// TIA Portal project "FactoryIO_Template_S7-1200_V15_V15.1" (V15.1)
// Vorlageprojekt für das Buch mit Zielsystem S7-1200

(* hardware
DEVICE "S7-1200 station_2"  S7-1200 Station
   slot 0: "Rack_0"  S7-1200 Rack  Rack  V1.0
   slot 1: "PLC_1"  CPU 1215C DC/DC/DC  6ES7 215-1AG40-0XB0  V4.2
   slot 2: "DI 16x24VDC_1"  6ES7 221-1BH32-0XB0  V2.0
   slot 3: "DQ 16x24VDC_1"  SM 1222 DQ16 x 24VDC  6ES7 222-1BH32-0XB0  V2.0
DEVICE "HMI_1"  TP1200 Comfort
   slot 0: "HMI_1"  TP1200 Comfort  6AV2 124-0MC01-0AX0  15.1.0.0
   slot 1: "HMI_RT_1"  TP1200 Comfort  6AV2 124-0MC01-0AX0  15.1.0.0
   slot 5: "HMI_1.IE_CP_1"  PROFINET Interface  15.0.1.0
      slot 1: "PROFINET Interface_1"  PROFINET Interface
         slot 1: "Port_1"  Port
         slot 2: "Port_2"  Port
   slot 7: "HMI_1.MPI/DP_CP_1"  MPI/DP Interface  15.0.1.0
*)

// ===== PLC "PLC_1"  CPU 1215C DC/DC/DC =====

VAR_GLOBAL   // PLC tag table "Default tag table"
   "Green Base Conv_Timer" AT %M5.6 : Bool;
   "Green Lid Conv_Timer" AT %M5.7 : Bool;
   "Metal Base Conv_Timer" AT %M6.0 : Bool;
   "Metal Lid Conv_Timer" AT %M6.1 : Bool;
   "Blue Base Conv_Timer" AT %M6.2 : Bool;
   "Blue Lid Conv_Timer" AT %M6.3 : Bool;
   "RESET_Conv_Timers" AT %M6.4 : Bool;
   "Emitter_Emit" AT %Q4.7 : Bool;
   "Emitter_Part" AT %QD30 : DInt;
   "Counter_Reset" AT %M6.5 : Bool;
   "n_trig[4]" AT %M5.5 : Bool;
   "at load" AT %I13.5 : Bool;
   "left" AT %Q5.2 : Bool;
   "right" AT %Q5.3 : Bool;
   "lift" AT %Q5.4 : Bool;
   "targeted position" AT %QD34 : DInt;
   "at unload" AT %I13.7 : Bool;
   "moving x" AT %I14.0 : Bool;
   "moving z" AT %I14.1 : Bool;
   "at right" AT %I14.2 : Bool;
   "at left" AT %I14.3 : Bool;
   "at middle" AT %I14.4 : Bool;
   "shelf value" AT %MW46 : Word;
   "at entry" AT %I14.5 : Bool;
   "at exit" AT %I14.6 : Bool;
   "entry conveyor(1)" AT %Q5.5 : Bool;
   "loading coneyor" AT %Q5.6 : Bool;
   "unloading coneyor" AT %Q5.7 : Bool;
   "exit conveyor" AT %Q6.0 : Bool;
   "FactoryIo_BugFix" AT %I14.7 : Bool;
   "Box Timing Temp" AT %M6.7 : Bool;
   "Boxes Emitter" AT %Q5.1 : Bool;
   "Boxes Conevyor" AT %Q5.0 : Bool;
   "Product Near Box" AT %I13.6 : Bool;
   "M11" AT %MD60 : DInt;
   "M22" AT %MD64 : DInt;
   "M33" AT %MD68 : DInt;
   "M44" AT %MD72 : DInt;
   "M55" AT %MD76 : DInt;
   "M66" AT %MD80 : DInt;
   "cont sinsor1" AT %I15.0 : Bool;
   "cont sinsor2" AT %I15.1 : Bool;
   "cont sinsor3" AT %I15.2 : Bool;
   "M77" AT %MD88 : DInt;
   "M88" AT %MD92 : DInt;
   "M99" AT %MD96 : DInt;
   "resat" AT %M100.0 : Bool;
   "M110" AT %MD110 : DInt;
   "M120" AT %MD114 : DInt;
   "M130" AT %MD118 : DInt;
   "HMI_UNLOAD" AT %I122.0 : Bool;
END_VAR

VAR_GLOBAL   // PLC tag table "Default tag table_1"
   "ntrig3" AT %M0.4 : Bool;
   "Sorter Memory" AT %MW2 : Word;
   "Metal Base Belt" AT %Q1.1 : Bool;
   "Metal Lid Belt" AT %Q1.2 : Bool;
   "Green Base Belt" AT %Q1.3 : Bool;
   "Green Lid Belt" AT %Q1.4 : Bool;
   "Blue Base Belt" AT %Q1.5 : Bool;
   "Blue Lid Belt" AT %Q1.6 : Bool;
   "#p_trig[0]" AT %M1.7 : Bool;
   "#p_trig[1]" AT %M4.0 : Bool;
   "#p_trig[2]" AT %M4.1 : Bool;
   "#p_trig[3]" AT %M4.2 : Bool;
   "Lid at place" AT %M4.3 : Bool;
   "Lid Clamped" AT %M4.4 : Bool;
   "Two_Axis_Sequence_Done" AT %M4.5 : Bool;
   "Clamp_Lid" AT %M4.6 : Bool;
   "Raise_Lid" AT %M4.7 : Bool;
   "MB_Available" AT %I10.2 : Bool;
   "ML_Available" AT %I10.3 : Bool;
   "GB_Available" AT %I10.4 : Bool;
   "GL_Available" AT %I10.5 : Bool;
   "BB_Available" AT %I10.6 : Bool;
   "BL_Available" AT %I10.7 : Bool;
   "Metal Base Clamp_Positioned" AT %I11.0 : Bool;
   "Metal Lid Clamp_Positioned" AT %I11.1 : Bool;
   "Green Base Clamp_Positioned" AT %I11.2 : Bool;
   "Green Lid Clamp_Positioned" AT %I11.3 : Bool;
   "Blue Base Clamp_Positioned" AT %I11.4 : Bool;
   "Blue Lid Clamp_Positioned" AT %I11.5 : Bool;
   "Metal Lid C_Conv" AT %Q2.5 : Bool;
   "Metal Base C_Conv" AT %Q2.6 : Bool;
   "Green Lid C_Conv" AT %Q2.7 : Bool;
   "Green Base C_Conv" AT %Q3.0 : Bool;
   "Blue Lid C_Conv" AT %Q3.1 : Bool;
   "Blue Base C_Conv" AT %Q3.2 : Bool;
   "Metal Lid (Clamped)" AT %I11.6 : Bool;
   "Metal Base (Clamped)" AT %I11.7 : Bool;
   "Green Lid (Clamped)" AT %I12.0 : Bool;
   "Green Base (Clamped)" AT %I12.1 : Bool;
   "Blue Lid (Clamped)" AT %I12.2 : Bool;
   "Blue Base (Clamped)" AT %I12.3 : Bool;
   "ML (Clamp)" AT %Q1.7 : Bool;
   "MB (Clamp)" AT %Q2.0 : Bool;
   "GL (Clamp)" AT %Q2.1 : Bool;
   "GB (Clamp)" AT %Q2.2 : Bool;
   "BL (Clamp)" AT %Q2.3 : Bool;
   "BB (Clamp)" AT %Q2.4 : Bool;
   "Metal Piece (Raise)" AT %Q3.3 : Bool;
   "Green Piece (Raise)" AT %Q3.4 : Bool;
   "Blue Piece (Raise)" AT %Q3.5 : Bool;
   "Moving X1" AT %I12.4 : Bool;
   "Moving Z1" AT %I12.5 : Bool;
   "Moving X2" AT %I12.6 : Bool;
   "Moving Z2" AT %I12.7 : Bool;
   "Moving X3" AT %I13.0 : Bool;
   "Moving Z3" AT %I13.1 : Bool;
   "Grab1" AT %Q4.4 : Bool;
   "Grab2" AT %Q4.5 : Bool;
   "Grab3" AT %Q4.6 : Bool;
   "Move X1" AT %Q3.6 : Bool;
   "Move Z1" AT %Q3.7 : Bool;
   "Move X2" AT %Q4.0 : Bool;
   "Move Z2" AT %Q4.1 : Bool;
   "Move X3" AT %Q4.2 : Bool;
   "Move Z3" AT %Q4.3 : Bool;
   "Two_Axis_Sequence_Done1" AT %M0.5 : Bool;
   "Two_Axis_Sequence_Done2" AT %M0.6 : Bool;
   "Two_Axis_Sequence_Done3" AT %M0.7 : Bool;
   "Item_Detected1" AT %I13.2 : Bool;
   "Item_Detected2" AT %I13.3 : Bool;
   "Item_Detected3" AT %I13.4 : Bool;
   "ML C Latch" AT %M1.0 : Bool;
   "MB C Latch" AT %M1.1 : Bool;
   "GL C Latch" AT %M1.2 : Bool;
   "GB C Latch" AT %M1.3 : Bool;
   "BL C Latch" AT %M1.4 : Bool;
   "BB C Latch" AT %M1.5 : Bool;
   "RESET_METAL" AT %M1.6 : Bool;
   "RESET_GREEN" AT %M5.0 : Bool;
   "RESET_BLUE" AT %M5.1 : Bool;
   "Tag_1" AT %M10.7 : Bool;
   "Tag_2" AT %M5.3 : Bool;
   "Tag_3" AT %M5.4 : Bool;
END_VAR

VAR_GLOBAL CONSTANT   // PLC tag table "Default tag table_1"
   "None(1)" : Pip := 65535;
   "Automatic update(1)" : Pip := 0;
   "PIP 1(1)" : Pip := 1;
   "PIP 2(1)" : Pip := 2;
   "PIP 3(1)" : Pip := 3;
   "PIP 4(1)" : Pip := 4;
   "PIP OB Servo(1)" : Pip := 32768;
   "Local~MC(2)" : Hw_SubModule := 51;
   "Local~Common(2)" : Hw_SubModule := 50;
   "Local~Device(2)" : Hw_Device := 32;
   "Local~Configuration(2)" : Hw_SubModule := 33;
   "Local~Exec(2)" : Hw_SubModule := 52;
   "Local(2)" : Hw_SubModule := 49;
   "Local~PROFINET_interface_1(1)" : Hw_Interface := 64;
   "Local~PROFINET_interface_1~Port_1(1)" : Hw_Interface := 65;
   "Local~PROFINET_interface_1~Port_2(1)" : Hw_Interface := 66;
   "Local~HSC_1(2)" : Hw_Hsc := 257;
   "Local~HSC_2(2)" : Hw_Hsc := 258;
   "Local~HSC_3(2)" : Hw_Hsc := 259;
   "Local~HSC_4(2)" : Hw_Hsc := 260;
   "Local~HSC_5(2)" : Hw_Hsc := 261;
   "Local~HSC_6(2)" : Hw_Hsc := 262;
   "Local~AI_2_AQ_2_1(1)" : Hw_SubModule := 263;
   "Local~DI_14_DQ_10_1(1)" : Hw_SubModule := 264;
   "Local~Pulse_1(2)" : Hw_Pwm := 265;
   "Local~Pulse_2(2)" : Hw_Pwm := 266;
   "Local~Pulse_3(2)" : Hw_Pwm := 267;
   "Local~Pulse_4(2)" : Hw_Pwm := 268;
   "OB_Main(2)" : OB_PCYCLE := 1;
   "Local~DI_16x24VDC_1(1)" : Hw_SubModule := 269;
   "Local~DQ_8x24VDC__1" : Hw_SubModule := 270;
END_VAR

VAR_GLOBAL   // PLC tag table "Standard-Variablentabelle"
   "Entry Conveyor Stop" AT %M0.0 : Bool;
   "ntrig0" AT %M0.1 : Bool;
   "Stop Sensor 1" AT %I10.0 : Bool;
   "Stop Sensor 2" AT %I10.1 : Bool;
   "ntrig1" AT %M0.2 : Bool;
   "Sorting Conveyor 1" AT %Q0.7 : Bool;
   "Sorting Conveyor 2" AT %Q1.0 : Bool;
   "ntrig2" AT %M0.3 : Bool;
END_VAR

VAR_GLOBAL CONSTANT   // PLC tag table "Standard-Variablentabelle"
   "Keiner" : Pip := 65535;
   "Automatische Aktualisierung" : Pip := 0;
   "TPA 1" : Pip := 1;
   "TPA 2" : Pip := 2;
   "TPA 3" : Pip := 3;
   "TPA 4" : Pip := 4;
   "TPA OB Servo" : Pip := 32768;
   "Local~MC(1)" : Hw_SubModule := 51;
   "Local~Common(1)" : Hw_SubModule := 50;
   "Local~Device(1)" : Hw_Device := 32;
   "Local~Configuration(1)" : Hw_SubModule := 33;
   "Local~Exec(1)" : Hw_SubModule := 52;
   "Local(1)" : Hw_SubModule := 49;
   "Local~PROFINET-Schnittstelle_1" : Hw_Interface := 64;
   "Local~PROFINET-Schnittstelle_1~Port_1" : Hw_Interface := 65;
   "Local~HSC_1(1)" : Hw_Hsc := 257;
   "Local~HSC_2(1)" : Hw_Hsc := 258;
   "Local~HSC_3(1)" : Hw_Hsc := 259;
   "Local~HSC_4(1)" : Hw_Hsc := 260;
   "Local~HSC_5(1)" : Hw_Hsc := 261;
   "Local~HSC_6(1)" : Hw_Hsc := 262;
   "Local~AI_2_1" : Hw_SubModule := 263;
   "Local~DI_6_DQ_4_1" : Hw_SubModule := 264;
   "Local~Pulse_1(1)" : Hw_Pwm := 265;
   "Local~Pulse_2(1)" : Hw_Pwm := 266;
   "Local~Pulse_3(1)" : Hw_Pwm := 267;
   "Local~Pulse_4(1)" : Hw_Pwm := 268;
   "OB_Main(1)" : OB_PCYCLE := 1;
END_VAR

VAR_GLOBAL   // PLC tag table "Tag table from XML_1"
   "Entry Conveyor" AT %Q0.0 : Bool;
   "Metal Base Arm" AT %Q0.1 : Bool;
   "Metal Lid Arm" AT %Q0.2 : Bool;
   "Green Base Arm" AT %Q0.3 : Bool;
   "Green Lid Arm" AT %Q0.4 : Bool;
   "Blue Base Arm" AT %Q0.5 : Bool;
   "Blue Lid Arm" AT %Q0.6 : Bool;
   "Vision Sensor 1 (Value)" AT %ID30 : DInt;
END_VAR

DATA_BLOCK "Pick&Place_DB"   // DB2
{ S7_Optimized_Access := 'TRUE' }
VERSION : 0.1
// stored: InstanceOfName Pick&Place
"Pick&Place"
BEGIN
END_DATA_BLOCK

DATA_BLOCK "Base_Conveyor_DB"   // DB3
{ S7_Optimized_Access := 'TRUE' }
VERSION : 0.1
// stored: InstanceOfName Base_Conveyor
"Base_Conveyor"
BEGIN
END_DATA_BLOCK

DATA_BLOCK "Base_Conveyor_DB_1"   // DB4
{ S7_Optimized_Access := 'TRUE' }
VERSION : 0.1
// stored: InstanceOfName Base_Conveyor
"Base_Conveyor"
BEGIN
END_DATA_BLOCK

DATA_BLOCK "Base_Conveyor_DB_2"   // DB5
{ S7_Optimized_Access := 'TRUE' }
VERSION : 0.1
// stored: InstanceOfName Base_Conveyor
"Base_Conveyor"
BEGIN
END_DATA_BLOCK

DATA_BLOCK "Lids_Conveyor_DB"   // DB6
{ S7_Optimized_Access := 'TRUE' }
VERSION : 0.1
// stored: InstanceOfName Lids_Conveyor
"Lids_Conveyor"
BEGIN
END_DATA_BLOCK

DATA_BLOCK "Lids_Conveyor_DB_1"   // DB7
{ S7_Optimized_Access := 'TRUE' }
VERSION : 0.1
// stored: InstanceOfName Lids_Conveyor
"Lids_Conveyor"
BEGIN
END_DATA_BLOCK

DATA_BLOCK "Lids_Conveyor_DB_2"   // DB8
{ S7_Optimized_Access := 'TRUE' }
VERSION : 0.1
// stored: InstanceOfName Lids_Conveyor
"Lids_Conveyor"
BEGIN
END_DATA_BLOCK

DATA_BLOCK "Clamp_Base1"   // DB9
{ S7_Optimized_Access := 'TRUE' }
VERSION : 0.1
// stored: InstanceOfName Clamp
"Clamp"
BEGIN
END_DATA_BLOCK

DATA_BLOCK "Clamp_Base2"   // DB10
{ S7_Optimized_Access := 'TRUE' }
VERSION : 0.1
// stored: InstanceOfName Clamp
"Clamp"
BEGIN
END_DATA_BLOCK

DATA_BLOCK "Clamp_Base3"   // DB11
{ S7_Optimized_Access := 'TRUE' }
VERSION : 0.1
// stored: InstanceOfName Clamp
"Clamp"
BEGIN
END_DATA_BLOCK

DATA_BLOCK "Clamp_lid1"   // DB12
{ S7_Optimized_Access := 'TRUE' }
VERSION : 0.1
// stored: InstanceOfName Clamp
"Clamp"
BEGIN
END_DATA_BLOCK

DATA_BLOCK "Clamp_lid2"   // DB13
{ S7_Optimized_Access := 'TRUE' }
VERSION : 0.1
// stored: InstanceOfName Clamp
"Clamp"
BEGIN
END_DATA_BLOCK

DATA_BLOCK "Clamp_lid3"   // DB14
{ S7_Optimized_Access := 'TRUE' }
VERSION : 0.1
// stored: InstanceOfName Clamp
"Clamp"
BEGIN
END_DATA_BLOCK

DATA_BLOCK "Pick&Place_DB_1"   // DB15
{ S7_Optimized_Access := 'TRUE' }
VERSION : 0.1
// stored: InstanceOfName Pick&Place
"Pick&Place"
BEGIN
END_DATA_BLOCK

DATA_BLOCK "Pick&Place_DB_2"   // DB16
{ S7_Optimized_Access := 'TRUE' }
VERSION : 0.1
// stored: InstanceOfName Pick&Place
"Pick&Place"
BEGIN
END_DATA_BLOCK

DATA_BLOCK "Pick&Place_DB_3"   // DB17
{ S7_Optimized_Access := 'TRUE' }
VERSION : 0.1
// stored: InstanceOfName Pick&Place
"Pick&Place"
BEGIN
END_DATA_BLOCK

DATA_BLOCK "Block_1_DB"   // DB24
{ S7_Optimized_Access := 'TRUE' }
VERSION : 0.1
// stored: InstanceOfName Block_1
"Block_1"
BEGIN
END_DATA_BLOCK

DATA_BLOCK "Block_1_DB_1"   // DB25
{ S7_Optimized_Access := 'TRUE' }
VERSION : 0.1
// stored: InstanceOfName Block_1
"Block_1"
BEGIN
END_DATA_BLOCK

DATA_BLOCK "Block_2_DB"   // DB26
{ S7_Optimized_Access := 'TRUE' }
VERSION : 0.1
// stored: InstanceOfName Block_2
"Block_2"
BEGIN
END_DATA_BLOCK

DATA_BLOCK "Block_1_DB_2"   // DB27
{ S7_Optimized_Access := 'TRUE' }
VERSION : 0.1
// stored: InstanceOfName Block_1
"Block_1"
BEGIN
END_DATA_BLOCK

// folder: System blocks/Program resources

DATA_BLOCK "IEC_Timer_0_DB"   // DB1
{ S7_Optimized_Access := 'TRUE' }
AUTHOR : Simatic
FAMILY : IEC
NAME : IEC_TMR
VERSION : 1.0
// stored: InstanceOfName IEC_TIMER
"IEC_TIMER"
BEGIN
END_DATA_BLOCK

DATA_BLOCK "IEC_Timer_0_DB_1"   // DB18
{ S7_Optimized_Access := 'TRUE' }
AUTHOR : Simatic
FAMILY : IEC
NAME : IEC_TMR
VERSION : 1.0
// stored: InstanceOfName IEC_TIMER
"IEC_TIMER"
BEGIN
END_DATA_BLOCK

DATA_BLOCK "IEC_Timer_0_DB_2"   // DB19
{ S7_Optimized_Access := 'TRUE' }
AUTHOR : Simatic
FAMILY : IEC
NAME : IEC_TMR
VERSION : 1.0
// stored: InstanceOfName IEC_TIMER
"IEC_TIMER"
BEGIN
END_DATA_BLOCK

DATA_BLOCK "IEC_Timer_0_DB_3"   // DB20
{ S7_Optimized_Access := 'TRUE' }
AUTHOR : Simatic
FAMILY : IEC
NAME : IEC_TMR
VERSION : 1.0
// stored: InstanceOfName IEC_TIMER
"IEC_TIMER"
BEGIN
END_DATA_BLOCK

DATA_BLOCK "IEC_Timer_0_DB_4"   // DB21
{ S7_Optimized_Access := 'TRUE' }
AUTHOR : Simatic
FAMILY : IEC
NAME : IEC_TMR
VERSION : 1.0
// stored: InstanceOfName IEC_TIMER
"IEC_TIMER"
BEGIN
END_DATA_BLOCK

DATA_BLOCK "IEC_Timer_0_DB_5"   // DB22
{ S7_Optimized_Access := 'TRUE' }
AUTHOR : Simatic
FAMILY : IEC
NAME : IEC_TMR
VERSION : 1.0
// stored: InstanceOfName IEC_TIMER
"IEC_TIMER"
BEGIN
END_DATA_BLOCK

DATA_BLOCK "IEC_Counter_0_DB[1]"   // DB23
{ S7_Optimized_Access := 'TRUE' }
AUTHOR : Simatic
FAMILY : IEC
NAME : CNTR
VERSION : 1.0
// stored: InstanceOfName IEC_COUNTER
"IEC_COUNTER"
BEGIN
END_DATA_BLOCK

DATA_BLOCK "IEC_Timer_0_DB_6"   // DB28
{ S7_Optimized_Access := 'TRUE' }
AUTHOR : Simatic
FAMILY : IEC
NAME : IEC_TMR
VERSION : 1.0
// stored: InstanceOfName IEC_TIMER
"IEC_TIMER"
BEGIN
END_DATA_BLOCK

DATA_BLOCK "IEC_Counter_0_DB"   // DB29
{ S7_Optimized_Access := 'TRUE' }
AUTHOR : Simatic
FAMILY : IEC
NAME : CNTR
VERSION : 1.0
// stored: InstanceOfName IEC_COUNTER
"IEC_COUNTER"
BEGIN
END_DATA_BLOCK

DATA_BLOCK "IEC_Counter_0_DB_1"   // DB30
{ S7_Optimized_Access := 'TRUE' }
AUTHOR : Simatic
FAMILY : IEC
NAME : CNTR
VERSION : 1.0
// stored: InstanceOfName IEC_COUNTER
"IEC_COUNTER"
BEGIN
END_DATA_BLOCK

DATA_BLOCK "IEC_Counter_0_DB_2"   // DB31
{ S7_Optimized_Access := 'TRUE' }
AUTHOR : Simatic
FAMILY : IEC
NAME : CNTR
VERSION : 1.0
// stored: InstanceOfName IEC_COUNTER
"IEC_COUNTER"
BEGIN
END_DATA_BLOCK

DATA_BLOCK "IEC_Counter_0_DB_3"   // DB32
{ S7_Optimized_Access := 'TRUE' }
AUTHOR : Simatic
FAMILY : IEC
NAME : CNTR
VERSION : 1.0
// stored: InstanceOfName IEC_COUNTER
"IEC_COUNTER"
BEGIN
END_DATA_BLOCK

DATA_BLOCK "IEC_Counter_0_DB_4"   // DB33
{ S7_Optimized_Access := 'TRUE' }
AUTHOR : Simatic
FAMILY : IEC
NAME : CNTR
VERSION : 1.0
// stored: InstanceOfName IEC_COUNTER
"IEC_COUNTER"
BEGIN
END_DATA_BLOCK

DATA_BLOCK "IEC_Counter_0_DB_5"   // DB34
{ S7_Optimized_Access := 'TRUE' }
AUTHOR : Simatic
FAMILY : IEC
NAME : CNTR
VERSION : 1.0
// stored: InstanceOfName IEC_COUNTER
"IEC_COUNTER"
BEGIN
END_DATA_BLOCK

DATA_BLOCK "IEC_Counter_0_DB_6"   // DB35
{ S7_Optimized_Access := 'TRUE' }
AUTHOR : Simatic
FAMILY : IEC
NAME : CNTR
VERSION : 1.0
// stored: InstanceOfName IEC_COUNTER
"IEC_COUNTER"
BEGIN
END_DATA_BLOCK

DATA_BLOCK "IEC_Counter_0_DB_7"   // DB36
{ S7_Optimized_Access := 'TRUE' }
AUTHOR : Simatic
FAMILY : IEC
NAME : CNTR
VERSION : 1.0
// stored: InstanceOfName IEC_COUNTER
"IEC_COUNTER"
BEGIN
END_DATA_BLOCK

DATA_BLOCK "IEC_Counter_0_DB_8"   // DB37
{ S7_Optimized_Access := 'TRUE' }
AUTHOR : Simatic
FAMILY : IEC
NAME : CNTR
VERSION : 1.0
// stored: InstanceOfName IEC_COUNTER
"IEC_COUNTER"
BEGIN
END_DATA_BLOCK

DATA_BLOCK "IEC_Counter_0_DB_9"   // DB38
{ S7_Optimized_Access := 'TRUE' }
AUTHOR : Simatic
FAMILY : IEC
NAME : CNTR
VERSION : 1.0
// stored: InstanceOfName IEC_COUNTER
"IEC_COUNTER"
BEGIN
END_DATA_BLOCK

DATA_BLOCK "IEC_Counter_0_DB_10"   // DB39
{ S7_Optimized_Access := 'TRUE' }
AUTHOR : Simatic
FAMILY : IEC
NAME : CNTR
VERSION : 1.0
// stored: InstanceOfName IEC_COUNTER
"IEC_COUNTER"
BEGIN
END_DATA_BLOCK

// folder: (top level)

FUNCTION_BLOCK "Clamp"   // FB1, LAD
{ S7_Optimized_Access := 'TRUE' }
VERSION : 0.1
   VAR_INPUT
      Start_Clamper_Sequence : Bool;
      Clamped_Sensor : Bool;
      Axis_Seq_Done : Bool;
   END_VAR
   VAR_OUTPUT
      Clamp : Bool;
      Raise_Clamp : Bool;
      Sequence_Done : Bool;
   END_VAR
   VAR
      Sequence_Active : Bool;
      Step1 : Int;
   END_VAR
   VAR RETAIN
      "TimeOn1.PT" : Int;
   END_VAR
   VAR
      "p_trig[1]" : Bool;
      "p_trig[0]" : Bool;
      "p_trig[2]" : Bool;
      "p_trig[3]" : Bool;
      Sequence_Done_Pulse : Bool;
      IEC_Timer_0_Instance : TON_TIME;
   END_VAR
   VAR_TEMP   // added for the SCL form of the ladder/FBD networks
      _w1 : Bool;
      _w2 : Bool;
      _w3 : Bool;
   END_VAR
BEGIN

REGION Network 1
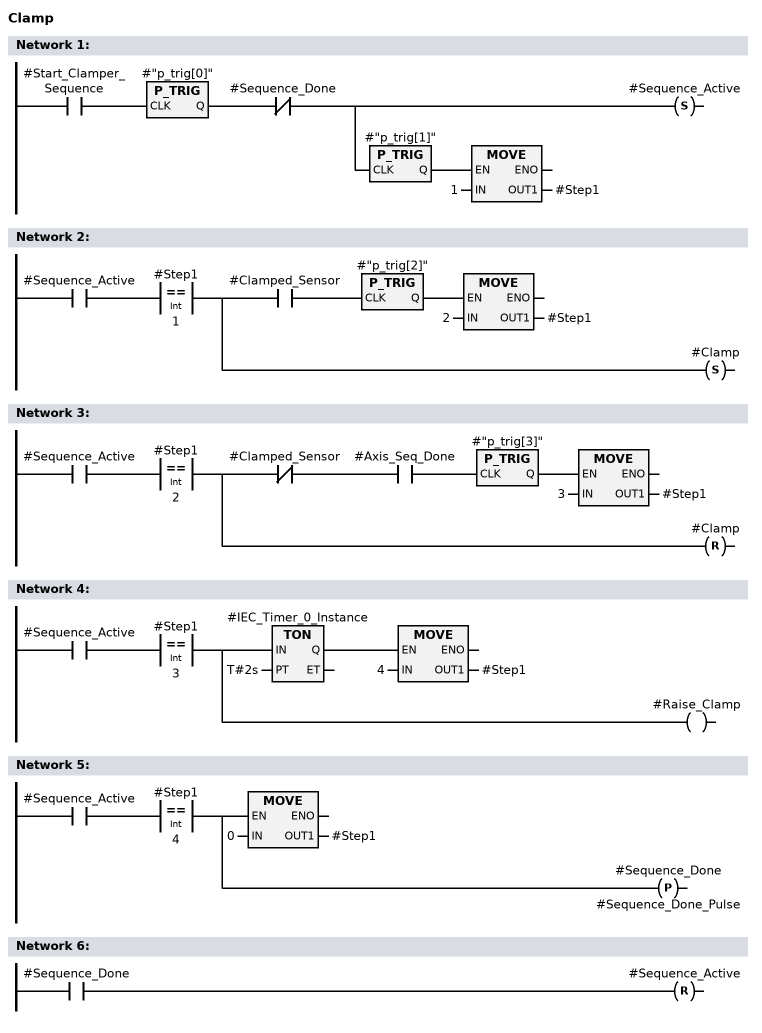
   RUNG wire#powerrail
      Contact( #Start_Clamper_Sequence )
      P_Trig( #"p_trig[0]" )
      I_Contact( #Sequence_Done )
      wire#w1
      S_Coil( #Sequence_Active )
   END_RUNG
   RUNG wire#w1
      P_Trig( #"p_trig[1]" )
      Move(in := 1, out1 => #Step1)
   END_RUNG
   // the same network as SCL:
   #_w1 := #Start_Clamper_Sequence AND NOT #"p_trig[0]";   // rising edge
   #"p_trig[0]" := #Start_Clamper_Sequence;
   #_w2 := #_w1 AND NOT #Sequence_Done;
   IF #_w2 THEN #Sequence_Active := TRUE; END_IF;
   #_w3 := #_w2 AND NOT #"p_trig[1]";   // rising edge
   #"p_trig[1]" := #_w2;
   IF #_w3 THEN #Step1 := 1; END_IF;
END_REGION

REGION Network 2
   RUNG wire#powerrail
      Contact( #Sequence_Active )
      { S7_Templates := "SrcType := Int" } EQ_Contact(in1 := #Step1, in2 := 1)
      wire#w1
      Contact( #Clamped_Sensor )
      P_Trig( #"p_trig[2]" )
      Move(in := 2, out1 => #Step1)
   END_RUNG
   RUNG wire#w1
      S_Coil( #Clamp )
   END_RUNG
   // the same network as SCL:
   #_w1 := #Sequence_Active AND (#Step1 = 1);
   #_w2 := #_w1 AND #Clamped_Sensor;
   #_w3 := #_w2 AND NOT #"p_trig[2]";   // rising edge
   #"p_trig[2]" := #_w2;
   IF #_w3 THEN #Step1 := 2; END_IF;
   IF #_w1 THEN #Clamp := TRUE; END_IF;
END_REGION

REGION Network 3
   RUNG wire#powerrail
      Contact( #Sequence_Active )
      { S7_Templates := "SrcType := Int" } EQ_Contact(in1 := #Step1, in2 := 2)
      wire#w1
      I_Contact( #Clamped_Sensor )
      Contact( #Axis_Seq_Done )
      P_Trig( #"p_trig[3]" )
      Move(in := 3, out1 => #Step1)
   END_RUNG
   RUNG wire#w1
      R_Coil( #Clamp )
   END_RUNG
   // the same network as SCL:
   #_w1 := #Sequence_Active AND (#Step1 = 2);
   #_w2 := #_w1 AND NOT #Clamped_Sensor AND #Axis_Seq_Done;
   #_w3 := #_w2 AND NOT #"p_trig[3]";   // rising edge
   #"p_trig[3]" := #_w2;
   IF #_w3 THEN #Step1 := 3; END_IF;
   IF #_w1 THEN #Clamp := FALSE; END_IF;
END_REGION

REGION Network 4
   #_w1 := #Sequence_Active AND (#Step1 = 3);
   #IEC_Timer_0_Instance(IN := #_w1, PT := T#2s);   // TON
   IF #IEC_Timer_0_Instance.Q THEN #Step1 := 4; END_IF;
   #Raise_Clamp := #_w1;
END_REGION

REGION Network 5
   #_w1 := #Sequence_Active AND (#Step1 = 4);
   IF #_w1 THEN #Step1 := 0; END_IF;
   #Sequence_Done := #_w1 AND NOT #Sequence_Done_Pulse;   // rising edge
   #Sequence_Done_Pulse := #_w1;
END_REGION

REGION Network 6
   RUNG wire#powerrail
      Contact( #Sequence_Done )
      R_Coil( #Sequence_Active )
   END_RUNG
   // the same network as SCL:
   IF #Sequence_Done THEN #Sequence_Active := FALSE; END_IF;
END_REGION
END_FUNCTION_BLOCK

FUNCTION_BLOCK "Pick&Place"   // FB2, LAD
{ S7_Optimized_Access := 'TRUE' }
VERSION : 0.1
   VAR_INPUT
      Start_Axis_Sequence : Bool;
      Moving_X : Bool;
      Moving_Z : Bool;
      Item_Detected : Bool;
   END_VAR
   VAR_OUTPUT
      Move_X : Bool;
      Move_Z : Bool;
      Item_Grab : Bool;
      RESET_CLAMP_COND : Bool;
      Sequence_Done : Bool;
   END_VAR
   VAR
      "n_trig[2]" : Bool;
      "n_trig[0]" : Bool;
      "n_trig[1]" : Bool;
      "Step" : Int;
      Sequence_Active : Bool;
      "p_trig[0]" : Bool;
      "p_trig[1]" : Bool;
      "p_trig[2]" : Bool;
      "n_trig[3]" : Bool;
      Sequence_Done_Pulses : Bool;
      "n_trig[4]" : Bool;
   END_VAR
   VAR_TEMP   // added for the SCL form of the ladder/FBD networks
      _w1 : Bool;
      _w2 : Bool;
      _w3 : Bool;
   END_VAR
BEGIN

REGION Network 1
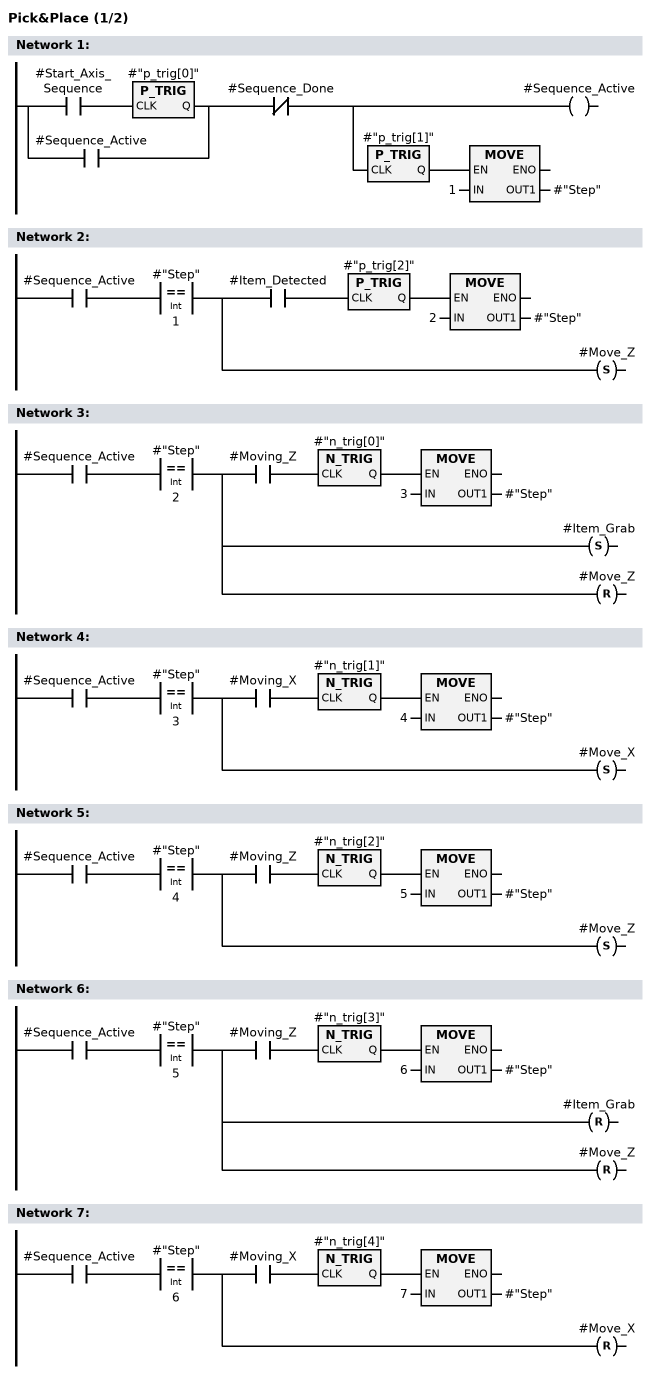
   RUNG wire#powerrail
      Contact( #Start_Axis_Sequence )
      P_Trig( #"p_trig[0]" )
      wire#w1
      I_Contact( #Sequence_Done )
      wire#w2
      Coil( #Sequence_Active )
   END_RUNG
   RUNG wire#powerrail
      Contact( #Sequence_Active )
   END_RUNG wire#w1
   RUNG wire#w2
      P_Trig( #"p_trig[1]" )
      Move(in := 1, out1 => #"Step")
   END_RUNG
   // the same network as SCL:
   #_w1 := #Start_Axis_Sequence AND NOT #"p_trig[0]";   // rising edge
   #"p_trig[0]" := #Start_Axis_Sequence;
   #Sequence_Active := (#_w1 OR #Sequence_Active) AND NOT #Sequence_Done;
   #_w2 := #Sequence_Active AND NOT #"p_trig[1]";   // rising edge
   #"p_trig[1]" := #Sequence_Active;
   IF #_w2 THEN #"Step" := 1; END_IF;
END_REGION

REGION Network 2
   RUNG wire#powerrail
      Contact( #Sequence_Active )
      { S7_Templates := "SrcType := Int" } EQ_Contact(in1 := #"Step", in2 := 1)
      wire#w1
      Contact( #Item_Detected )
      P_Trig( #"p_trig[2]" )
      Move(in := 2, out1 => #"Step")
   END_RUNG
   RUNG wire#w1
      S_Coil( #Move_Z )
   END_RUNG
   // the same network as SCL:
   #_w1 := #Sequence_Active AND (#"Step" = 1);
   #_w2 := #_w1 AND #Item_Detected;
   #_w3 := #_w2 AND NOT #"p_trig[2]";   // rising edge
   #"p_trig[2]" := #_w2;
   IF #_w3 THEN #"Step" := 2; END_IF;
   IF #_w1 THEN #Move_Z := TRUE; END_IF;
END_REGION

REGION Network 3
   RUNG wire#powerrail
      Contact( #Sequence_Active )
      { S7_Templates := "SrcType := Int" } EQ_Contact(in1 := #"Step", in2 := 2)
      wire#w1
      Contact( #Moving_Z )
      N_Trig( #"n_trig[0]" )
      Move(in := 3, out1 => #"Step")
   END_RUNG
   RUNG wire#w1
      S_Coil( #Item_Grab )
   END_RUNG
   RUNG wire#w1
      R_Coil( #Move_Z )
   END_RUNG
   // the same network as SCL:
   #_w1 := #Sequence_Active AND (#"Step" = 2);
   #_w2 := #_w1 AND #Moving_Z;
   #_w3 := NOT #_w2 AND #"n_trig[0]";   // falling edge
   #"n_trig[0]" := #_w2;
   IF #_w3 THEN #"Step" := 3; END_IF;
   IF #_w1 THEN
       #Item_Grab := TRUE;
       #Move_Z := FALSE;
   END_IF;
END_REGION

REGION Network 4
   RUNG wire#powerrail
      Contact( #Sequence_Active )
      { S7_Templates := "SrcType := Int" } EQ_Contact(in1 := #"Step", in2 := 3)
      wire#w1
      Contact( #Moving_X )
      N_Trig( #"n_trig[1]" )
      Move(in := 4, out1 => #"Step")
   END_RUNG
   RUNG wire#w1
      S_Coil( #Move_X )
   END_RUNG
   // the same network as SCL:
   #_w1 := #Sequence_Active AND (#"Step" = 3);
   #_w2 := #_w1 AND #Moving_X;
   #_w3 := NOT #_w2 AND #"n_trig[1]";   // falling edge
   #"n_trig[1]" := #_w2;
   IF #_w3 THEN #"Step" := 4; END_IF;
   IF #_w1 THEN #Move_X := TRUE; END_IF;
END_REGION

REGION Network 5
   RUNG wire#powerrail
      Contact( #Sequence_Active )
      { S7_Templates := "SrcType := Int" } EQ_Contact(in1 := #"Step", in2 := 4)
      wire#w1
      Contact( #Moving_Z )
      N_Trig( #"n_trig[2]" )
      Move(in := 5, out1 => #"Step")
   END_RUNG
   RUNG wire#w1
      S_Coil( #Move_Z )
   END_RUNG
   // the same network as SCL:
   #_w1 := #Sequence_Active AND (#"Step" = 4);
   #_w2 := #_w1 AND #Moving_Z;
   #_w3 := NOT #_w2 AND #"n_trig[2]";   // falling edge
   #"n_trig[2]" := #_w2;
   IF #_w3 THEN #"Step" := 5; END_IF;
   IF #_w1 THEN #Move_Z := TRUE; END_IF;
END_REGION

REGION Network 6
   RUNG wire#powerrail
      Contact( #Sequence_Active )
      { S7_Templates := "SrcType := Int" } EQ_Contact(in1 := #"Step", in2 := 5)
      wire#w1
      Contact( #Moving_Z )
      N_Trig( #"n_trig[3]" )
      Move(in := 6, out1 => #"Step")
   END_RUNG
   RUNG wire#w1
      R_Coil( #Item_Grab )
   END_RUNG
   RUNG wire#w1
      R_Coil( #Move_Z )
   END_RUNG
   // the same network as SCL:
   #_w1 := #Sequence_Active AND (#"Step" = 5);
   #_w2 := #_w1 AND #Moving_Z;
   #_w3 := NOT #_w2 AND #"n_trig[3]";   // falling edge
   #"n_trig[3]" := #_w2;
   IF #_w3 THEN #"Step" := 6; END_IF;
   IF #_w1 THEN
       #Item_Grab := FALSE;
       #Move_Z := FALSE;
   END_IF;
END_REGION

REGION Network 7
   RUNG wire#powerrail
      Contact( #Sequence_Active )
      { S7_Templates := "SrcType := Int" } EQ_Contact(in1 := #"Step", in2 := 6)
      wire#w1
      Contact( #Moving_X )
      N_Trig( #"n_trig[4]" )
      Move(in := 7, out1 => #"Step")
   END_RUNG
   RUNG wire#w1
      R_Coil( #Move_X )
   END_RUNG
   // the same network as SCL:
   #_w1 := #Sequence_Active AND (#"Step" = 6);
   #_w2 := #_w1 AND #Moving_X;
   #_w3 := NOT #_w2 AND #"n_trig[4]";   // falling edge
   #"n_trig[4]" := #_w2;
   IF #_w3 THEN #"Step" := 7; END_IF;
   IF #_w1 THEN #Move_X := FALSE; END_IF;
END_REGION

REGION Network 8
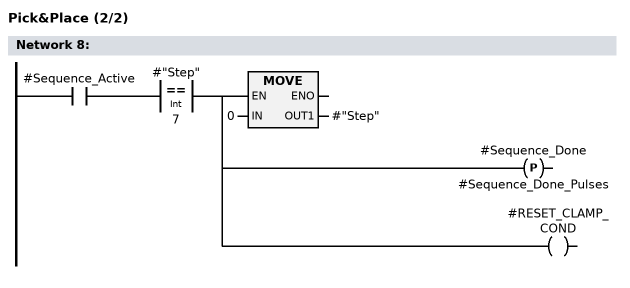
   #_w1 := #Sequence_Active AND (#"Step" = 7);
   IF #_w1 THEN #"Step" := 0; END_IF;
   #Sequence_Done := #_w1 AND NOT #Sequence_Done_Pulses;   // rising edge
   #Sequence_Done_Pulses := #_w1;
   #RESET_CLAMP_COND := #_w1;
END_REGION
END_FUNCTION_BLOCK

FUNCTION_BLOCK "Base_Conveyor"   // FB3, LAD
{ S7_Optimized_Access := 'TRUE' }
VERSION : 0.1
   VAR_INPUT
      Start_Bases_Conveyor : Bool;
      Stop_Bases_Conveyor : Bool;
   END_VAR
   VAR_OUTPUT
      Bases_Conveyor_Active : Bool;
   END_VAR
   VAR_TEMP
      "p_trig[0]" : Bool;
      "n_trig[0]" : Bool;
   END_VAR
   VAR_TEMP   // added for the SCL form of the ladder/FBD networks
      _w1 : Bool;
   END_VAR
BEGIN

REGION Network 1
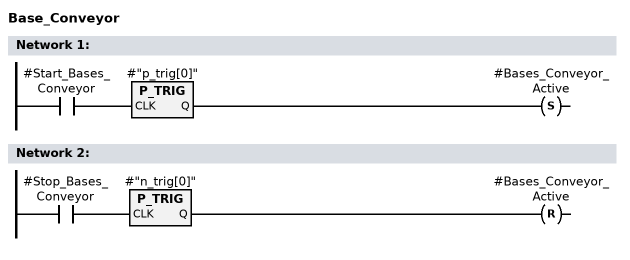
   RUNG wire#powerrail
      Contact( #Start_Bases_Conveyor )
      P_Trig( #"p_trig[0]" )
      S_Coil( #Bases_Conveyor_Active )
   END_RUNG
   // the same network as SCL:
   #_w1 := #Start_Bases_Conveyor AND NOT #"p_trig[0]";   // rising edge
   #"p_trig[0]" := #Start_Bases_Conveyor;
   IF #_w1 THEN #Bases_Conveyor_Active := TRUE; END_IF;
END_REGION

REGION Network 2
   RUNG wire#powerrail
      Contact( #Stop_Bases_Conveyor )
      P_Trig( #"n_trig[0]" )
      R_Coil( #Bases_Conveyor_Active )
   END_RUNG
   // the same network as SCL:
   #_w1 := #Stop_Bases_Conveyor AND NOT #"n_trig[0]";   // rising edge
   #"n_trig[0]" := #Stop_Bases_Conveyor;
   IF #_w1 THEN #Bases_Conveyor_Active := FALSE; END_IF;
END_REGION
END_FUNCTION_BLOCK

FUNCTION_BLOCK "Lids_Conveyor"   // FB4, LAD
{ S7_Optimized_Access := 'TRUE' }
VERSION : 0.1
   VAR_INPUT
      Start_Lids_Conveyor : Bool;
      Stop_Lids_Conveyor : Bool;
   END_VAR
   VAR_OUTPUT
      Lids_Conveyor_Active : Bool;
   END_VAR
   VAR_TEMP
      "p_trig[0]" : Bool;
      "n_trig[0]" : Bool;
   END_VAR
   VAR_TEMP   // added for the SCL form of the ladder/FBD networks
      _w1 : Bool;
   END_VAR
BEGIN

REGION Network 1
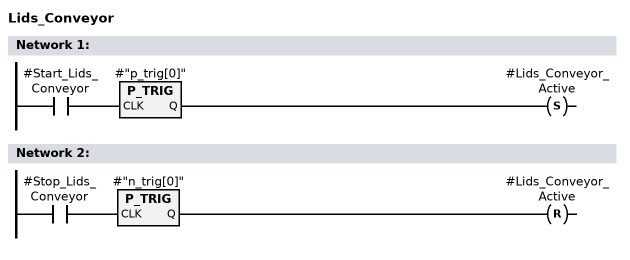
   RUNG wire#powerrail
      Contact( #Start_Lids_Conveyor )
      P_Trig( #"p_trig[0]" )
      S_Coil( #Lids_Conveyor_Active )
   END_RUNG
   // the same network as SCL:
   #_w1 := #Start_Lids_Conveyor AND NOT #"p_trig[0]";   // rising edge
   #"p_trig[0]" := #Start_Lids_Conveyor;
   IF #_w1 THEN #Lids_Conveyor_Active := TRUE; END_IF;
END_REGION

REGION Network 2
   RUNG wire#powerrail
      Contact( #Stop_Lids_Conveyor )
      P_Trig( #"n_trig[0]" )
      R_Coil( #Lids_Conveyor_Active )
   END_RUNG
   // the same network as SCL:
   #_w1 := #Stop_Lids_Conveyor AND NOT #"n_trig[0]";   // rising edge
   #"n_trig[0]" := #Stop_Lids_Conveyor;
   IF #_w1 THEN #Lids_Conveyor_Active := FALSE; END_IF;
END_REGION
END_FUNCTION_BLOCK

FUNCTION_BLOCK "Block_1"   // FB5, LAD
TITLE = stacker crane
{ S7_Optimized_Access := 'TRUE' }
VERSION : 0.1
   VAR_INPUT
      Start_Load_Sequence : Bool;
      Start_Unload_Sequence : Bool;
      "at right" : Bool;
      at_left : Bool;
      "at middle" : Bool;
      "moving X" : Bool;
      "moving Z" : Bool;
   END_VAR
   VAR_OUTPUT
      Stored_Shelf_Value : Int;
      forks_left : Bool;
      forks_right : Bool;
      lift : Bool;
      Unload_Sequence_Done : Bool;
      Load_Sequence_Done : Bool;
      target_position : Int;
   END_VAR
   VAR
      "n_trig[36]" : Bool;
      "n_trig[25]" : Bool;
      Unload_Sequence_Active : Bool;
      Load_Sequence_Active : Bool;
      p_trig25 : Bool;
      p_trig26 : Bool;
      p_trig27 : Bool;
      p_trig28 : Bool;
      "p_trig[29]" : Bool;
      n_trig35 : Bool;
      "n_trig[26]" : Bool;
      "n_trig[27]" : Bool;
      "n_tring[34]" : Bool;
      "n_trig[28]" : Bool;
      "n_trig[29]" : Bool;
      "n_trig[30]" : Bool;
      "n_trig[31]" : Bool;
      "n_trig[32]" : Bool;
      "n_trig[33]" : Bool;
      "pulse[5]" : Bool;
      "pulse[6]" : Bool;
      "Step" : Int;
   END_VAR
   VAR_TEMP   // added for the SCL form of the ladder/FBD networks
      _w1 : Bool;
      _w2 : Bool;
      _w3 : Bool;
   END_VAR
BEGIN

REGION Network 1: Load Sequence Active
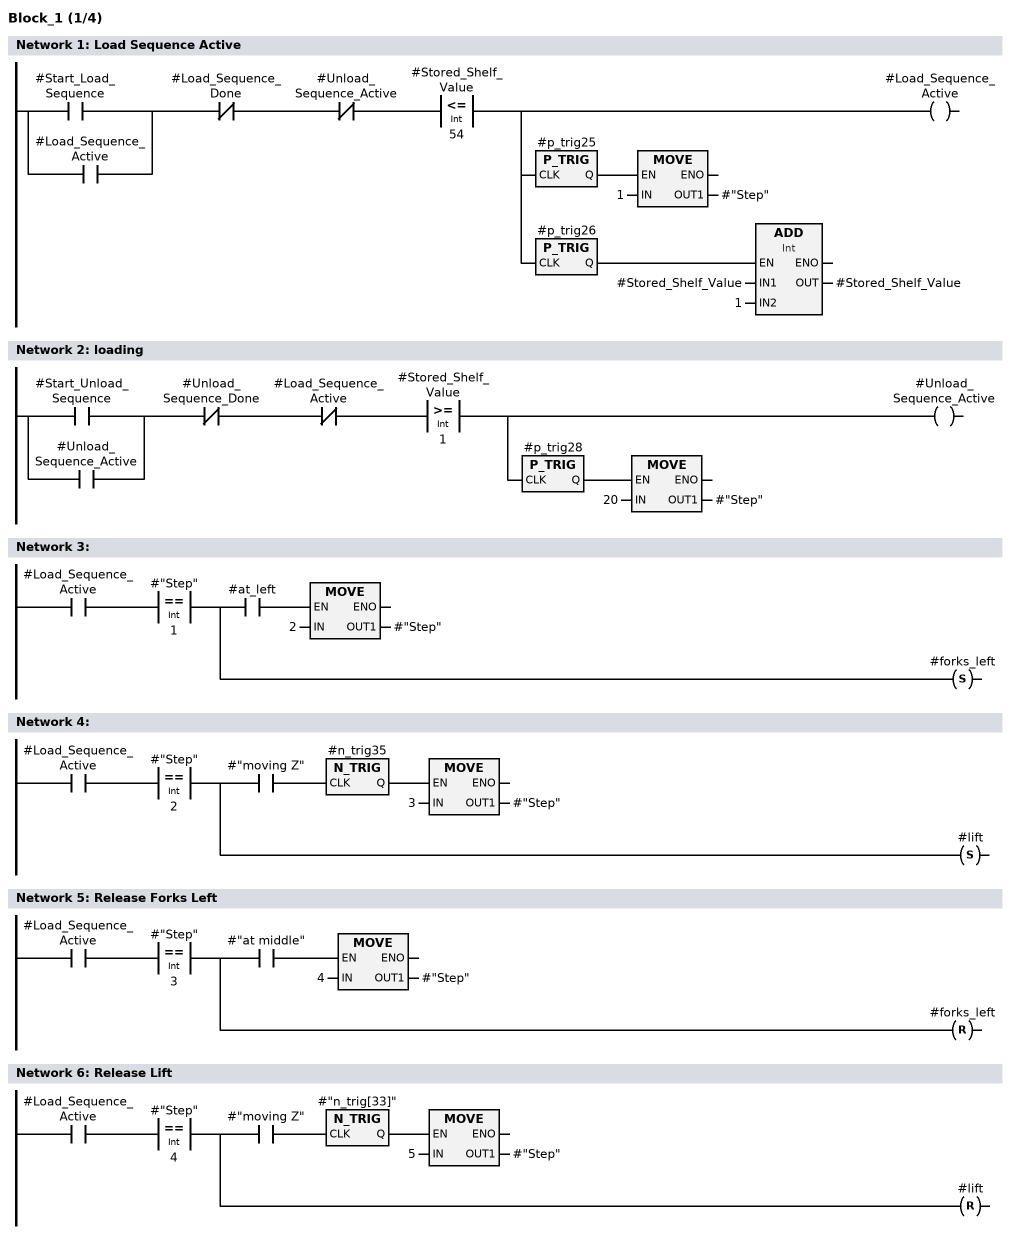
   RUNG wire#powerrail
      Contact( #Start_Load_Sequence )
      wire#w1
      I_Contact( #Load_Sequence_Done )
      I_Contact( #Unload_Sequence_Active )
      { S7_Templates := "SrcType := Int" } LE_Contact(in1 := #Stored_Shelf_Value, in2 := 54)
      wire#w2
      Coil( #Load_Sequence_Active )
   END_RUNG
   RUNG wire#powerrail
      Contact( #Load_Sequence_Active )
   END_RUNG wire#w1
   RUNG wire#w2
      P_Trig( #p_trig25 )
      Move(in := 1, out1 => #"Step")
   END_RUNG
   RUNG wire#w2
      P_Trig( #p_trig26 )
      { S7_Templates := "SrcType := Int" } Add(in1 := #Stored_Shelf_Value, in2 := 1, out => #Stored_Shelf_Value)
   END_RUNG
   // the same network as SCL:
   #Load_Sequence_Active := (#Start_Load_Sequence OR #Load_Sequence_Active) AND NOT #Load_Sequence_Done AND NOT #Unload_Sequence_Active AND (#Stored_Shelf_Value <= 54);
   #_w1 := #Load_Sequence_Active AND NOT #p_trig25;   // rising edge
   #p_trig25 := #Load_Sequence_Active;
   IF #_w1 THEN #"Step" := 1; END_IF;
   #_w2 := #Load_Sequence_Active AND NOT #p_trig26;   // rising edge
   #p_trig26 := #Load_Sequence_Active;
   IF #_w2 THEN #Stored_Shelf_Value := #Stored_Shelf_Value + 1; END_IF;
END_REGION

REGION Network 2: loading
   RUNG wire#powerrail
      Contact( #Start_Unload_Sequence )
      wire#w1
      I_Contact( #Unload_Sequence_Done )
      I_Contact( #Load_Sequence_Active )
      { S7_Templates := "SrcType := Int" } GE_Contact(in1 := #Stored_Shelf_Value, in2 := 1)
      wire#w2
      Coil( #Unload_Sequence_Active )
   END_RUNG
   RUNG wire#powerrail
      Contact( #Unload_Sequence_Active )
   END_RUNG wire#w1
   RUNG wire#w2
      P_Trig( #p_trig28 )
      Move(in := 20, out1 => #"Step")
   END_RUNG
   // the same network as SCL:
   #Unload_Sequence_Active := (#Start_Unload_Sequence OR #Unload_Sequence_Active) AND NOT #Unload_Sequence_Done AND NOT #Load_Sequence_Active AND (#Stored_Shelf_Value >= 1);
   #_w1 := #Unload_Sequence_Active AND NOT #p_trig28;   // rising edge
   #p_trig28 := #Unload_Sequence_Active;
   IF #_w1 THEN #"Step" := 20; END_IF;
END_REGION

REGION Network 3
   RUNG wire#powerrail
      Contact( #Load_Sequence_Active )
      { S7_Templates := "SrcType := Int" } EQ_Contact(in1 := #"Step", in2 := 1)
      wire#w1
      Contact( #at_left )
      Move(in := 2, out1 => #"Step")
   END_RUNG
   RUNG wire#w1
      S_Coil( #forks_left )
   END_RUNG
   // the same network as SCL:
   #_w1 := #Load_Sequence_Active AND (#"Step" = 1);
   IF #_w1 AND #at_left THEN #"Step" := 2; END_IF;
   IF #_w1 THEN #forks_left := TRUE; END_IF;
END_REGION

REGION Network 4
   RUNG wire#powerrail
      Contact( #Load_Sequence_Active )
      { S7_Templates := "SrcType := Int" } EQ_Contact(in1 := #"Step", in2 := 2)
      wire#w1
      Contact( #"moving Z" )
      N_Trig( #n_trig35 )
      Move(in := 3, out1 => #"Step")
   END_RUNG
   RUNG wire#w1
      S_Coil( #lift )
   END_RUNG
   // the same network as SCL:
   #_w1 := #Load_Sequence_Active AND (#"Step" = 2);
   #_w2 := #_w1 AND #"moving Z";
   #_w3 := NOT #_w2 AND #n_trig35;   // falling edge
   #n_trig35 := #_w2;
   IF #_w3 THEN #"Step" := 3; END_IF;
   IF #_w1 THEN #lift := TRUE; END_IF;
END_REGION

REGION Network 5: Release Forks Left
   RUNG wire#powerrail
      Contact( #Load_Sequence_Active )
      { S7_Templates := "SrcType := Int" } EQ_Contact(in1 := #"Step", in2 := 3)
      wire#w1
      Contact( #"at middle" )
      Move(in := 4, out1 => #"Step")
   END_RUNG
   RUNG wire#w1
      R_Coil( #forks_left )
   END_RUNG
   // the same network as SCL:
   #_w1 := #Load_Sequence_Active AND (#"Step" = 3);
   IF #_w1 AND #"at middle" THEN #"Step" := 4; END_IF;
   IF #_w1 THEN #forks_left := FALSE; END_IF;
END_REGION

REGION Network 6: Release Lift
   RUNG wire#powerrail
      Contact( #Load_Sequence_Active )
      { S7_Templates := "SrcType := Int" } EQ_Contact(in1 := #"Step", in2 := 4)
      wire#w1
      Contact( #"moving Z" )
      N_Trig( #"n_trig[33]" )
      Move(in := 5, out1 => #"Step")
   END_RUNG
   RUNG wire#w1
      R_Coil( #lift )
   END_RUNG
   // the same network as SCL:
   #_w1 := #Load_Sequence_Active AND (#"Step" = 4);
   #_w2 := #_w1 AND #"moving Z";
   #_w3 := NOT #_w2 AND #"n_trig[33]";   // falling edge
   #"n_trig[33]" := #_w2;
   IF #_w3 THEN #"Step" := 5; END_IF;
   IF #_w1 THEN #lift := FALSE; END_IF;
END_REGION

REGION Network 7: Counter For Storage & Move X position
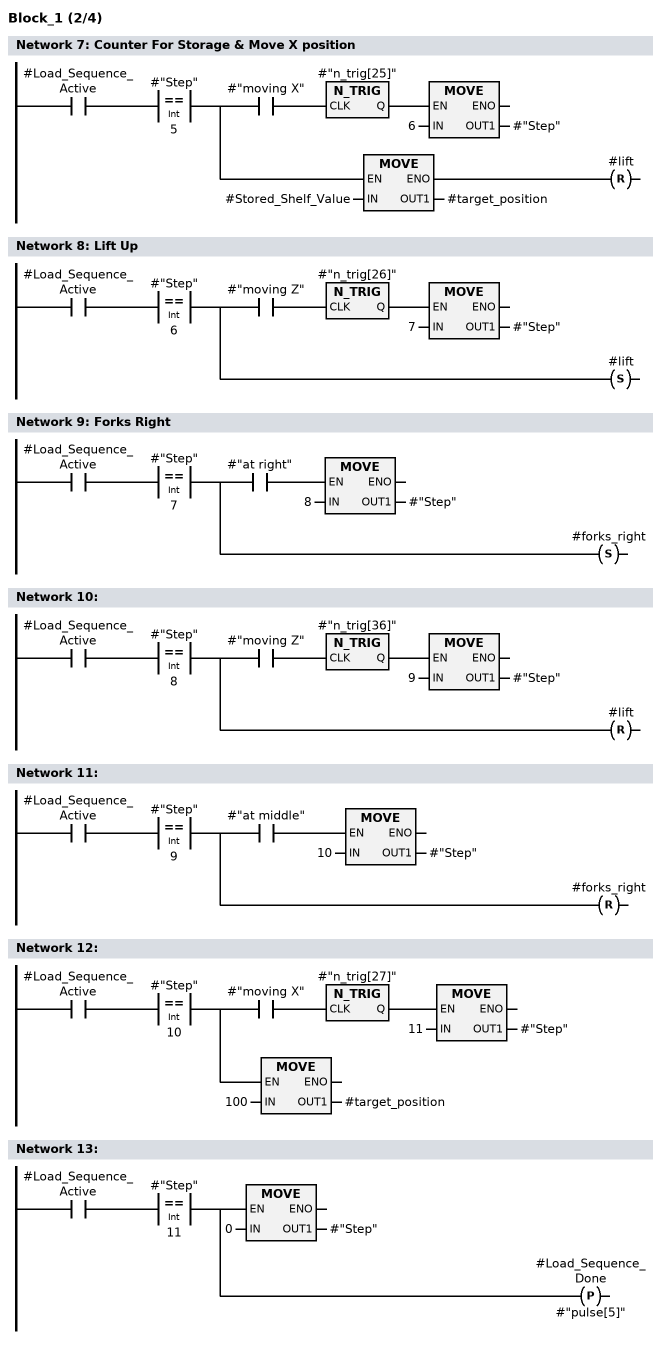
   RUNG wire#powerrail
      Contact( #Load_Sequence_Active )
      { S7_Templates := "SrcType := Int" } EQ_Contact(in1 := #"Step", in2 := 5)
      wire#w1
      Contact( #"moving X" )
      N_Trig( #"n_trig[25]" )
      Move(in := 6, out1 => #"Step")
   END_RUNG
   RUNG wire#w1
      Move(in := #Stored_Shelf_Value, out1 => #target_position)
      R_Coil( #lift )
   END_RUNG
   // the same network as SCL:
   #_w1 := #Load_Sequence_Active AND (#"Step" = 5);
   #_w2 := #_w1 AND #"moving X";
   #_w3 := NOT #_w2 AND #"n_trig[25]";   // falling edge
   #"n_trig[25]" := #_w2;
   IF #_w3 THEN #"Step" := 6; END_IF;
   IF #_w1 THEN
       #target_position := #Stored_Shelf_Value;
       #lift := FALSE;
   END_IF;
END_REGION

REGION Network 8: Lift Up
   RUNG wire#powerrail
      Contact( #Load_Sequence_Active )
      { S7_Templates := "SrcType := Int" } EQ_Contact(in1 := #"Step", in2 := 6)
      wire#w1
      Contact( #"moving Z" )
      N_Trig( #"n_trig[26]" )
      Move(in := 7, out1 => #"Step")
   END_RUNG
   RUNG wire#w1
      S_Coil( #lift )
   END_RUNG
   // the same network as SCL:
   #_w1 := #Load_Sequence_Active AND (#"Step" = 6);
   #_w2 := #_w1 AND #"moving Z";
   #_w3 := NOT #_w2 AND #"n_trig[26]";   // falling edge
   #"n_trig[26]" := #_w2;
   IF #_w3 THEN #"Step" := 7; END_IF;
   IF #_w1 THEN #lift := TRUE; END_IF;
END_REGION

REGION Network 9: Forks Right
   RUNG wire#powerrail
      Contact( #Load_Sequence_Active )
      { S7_Templates := "SrcType := Int" } EQ_Contact(in1 := #"Step", in2 := 7)
      wire#w1
      Contact( #"at right" )
      Move(in := 8, out1 => #"Step")
   END_RUNG
   RUNG wire#w1
      S_Coil( #forks_right )
   END_RUNG
   // the same network as SCL:
   #_w1 := #Load_Sequence_Active AND (#"Step" = 7);
   IF #_w1 AND #"at right" THEN #"Step" := 8; END_IF;
   IF #_w1 THEN #forks_right := TRUE; END_IF;
END_REGION

REGION Network 10
   RUNG wire#powerrail
      Contact( #Load_Sequence_Active )
      { S7_Templates := "SrcType := Int" } EQ_Contact(in1 := #"Step", in2 := 8)
      wire#w1
      Contact( #"moving Z" )
      N_Trig( #"n_trig[36]" )
      Move(in := 9, out1 => #"Step")
   END_RUNG
   RUNG wire#w1
      R_Coil( #lift )
   END_RUNG
   // the same network as SCL:
   #_w1 := #Load_Sequence_Active AND (#"Step" = 8);
   #_w2 := #_w1 AND #"moving Z";
   #_w3 := NOT #_w2 AND #"n_trig[36]";   // falling edge
   #"n_trig[36]" := #_w2;
   IF #_w3 THEN #"Step" := 9; END_IF;
   IF #_w1 THEN #lift := FALSE; END_IF;
END_REGION

REGION Network 11
   RUNG wire#powerrail
      Contact( #Load_Sequence_Active )
      { S7_Templates := "SrcType := Int" } EQ_Contact(in1 := #"Step", in2 := 9)
      wire#w1
      Contact( #"at middle" )
      Move(in := 10, out1 => #"Step")
   END_RUNG
   RUNG wire#w1
      R_Coil( #forks_right )
   END_RUNG
   // the same network as SCL:
   #_w1 := #Load_Sequence_Active AND (#"Step" = 9);
   IF #_w1 AND #"at middle" THEN #"Step" := 10; END_IF;
   IF #_w1 THEN #forks_right := FALSE; END_IF;
END_REGION

REGION Network 12
   RUNG wire#powerrail
      Contact( #Load_Sequence_Active )
      { S7_Templates := "SrcType := Int" } EQ_Contact(in1 := #"Step", in2 := 10)
      wire#w1
      Contact( #"moving X" )
      N_Trig( #"n_trig[27]" )
      Move(in := 11, out1 => #"Step")
   END_RUNG
   RUNG wire#w1
      Move(in := 100, out1 => #target_position)
   END_RUNG
   // the same network as SCL:
   #_w1 := #Load_Sequence_Active AND (#"Step" = 10);
   #_w2 := #_w1 AND #"moving X";
   #_w3 := NOT #_w2 AND #"n_trig[27]";   // falling edge
   #"n_trig[27]" := #_w2;
   IF #_w3 THEN #"Step" := 11; END_IF;
   IF #_w1 THEN #target_position := 100; END_IF;
END_REGION

REGION Network 13
   #_w1 := #Load_Sequence_Active AND (#"Step" = 11);
   IF #_w1 THEN #"Step" := 0; END_IF;
   #Load_Sequence_Done := #_w1 AND NOT #"pulse[5]";   // rising edge
   #"pulse[5]" := #_w1;
END_REGION

REGION Network 14
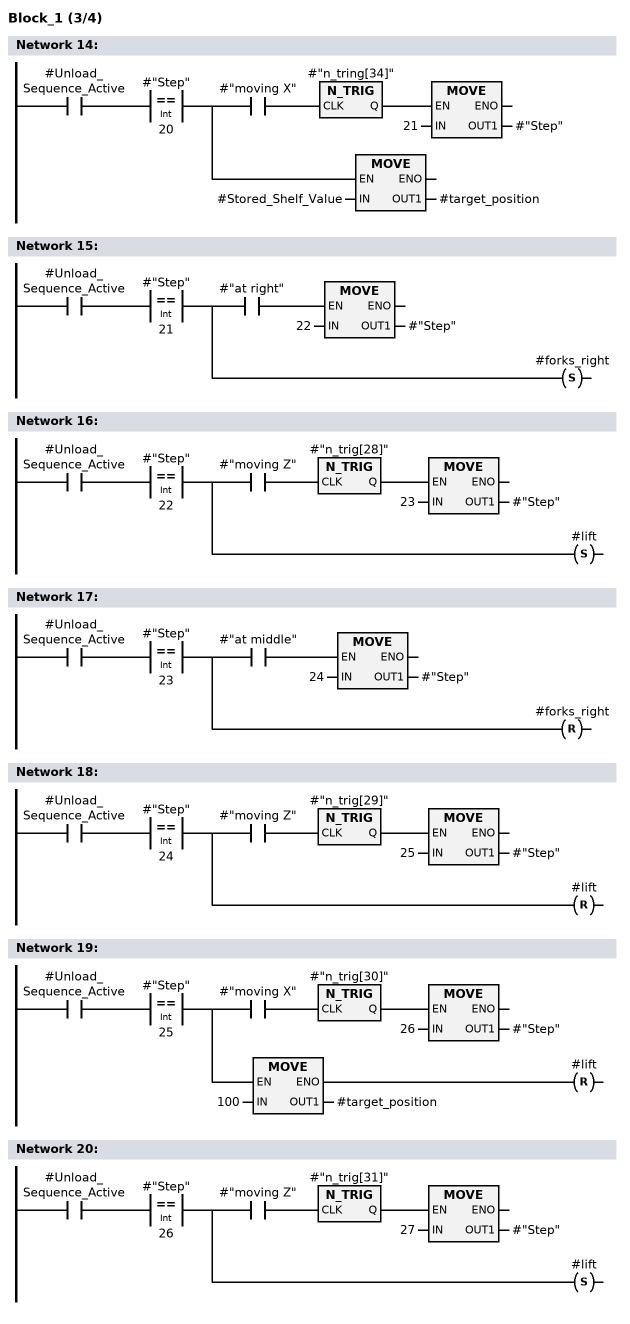
   RUNG wire#powerrail
      Contact( #Unload_Sequence_Active )
      { S7_Templates := "SrcType := Int" } EQ_Contact(in1 := #"Step", in2 := 20)
      wire#w1
      Contact( #"moving X" )
      N_Trig( #"n_tring[34]" )
      Move(in := 21, out1 => #"Step")
   END_RUNG
   RUNG wire#w1
      Move(in := #Stored_Shelf_Value, out1 => #target_position)
   END_RUNG
   // the same network as SCL:
   #_w1 := #Unload_Sequence_Active AND (#"Step" = 20);
   #_w2 := #_w1 AND #"moving X";
   #_w3 := NOT #_w2 AND #"n_tring[34]";   // falling edge
   #"n_tring[34]" := #_w2;
   IF #_w3 THEN #"Step" := 21; END_IF;
   IF #_w1 THEN #target_position := #Stored_Shelf_Value; END_IF;
END_REGION

REGION Network 15
   RUNG wire#powerrail
      Contact( #Unload_Sequence_Active )
      { S7_Templates := "SrcType := Int" } EQ_Contact(in1 := #"Step", in2 := 21)
      wire#w1
      Contact( #"at right" )
      Move(in := 22, out1 => #"Step")
   END_RUNG
   RUNG wire#w1
      S_Coil( #forks_right )
   END_RUNG
   // the same network as SCL:
   #_w1 := #Unload_Sequence_Active AND (#"Step" = 21);
   IF #_w1 AND #"at right" THEN #"Step" := 22; END_IF;
   IF #_w1 THEN #forks_right := TRUE; END_IF;
END_REGION

REGION Network 16
   RUNG wire#powerrail
      Contact( #Unload_Sequence_Active )
      { S7_Templates := "SrcType := Int" } EQ_Contact(in1 := #"Step", in2 := 22)
      wire#w1
      Contact( #"moving Z" )
      N_Trig( #"n_trig[28]" )
      Move(in := 23, out1 => #"Step")
   END_RUNG
   RUNG wire#w1
      S_Coil( #lift )
   END_RUNG
   // the same network as SCL:
   #_w1 := #Unload_Sequence_Active AND (#"Step" = 22);
   #_w2 := #_w1 AND #"moving Z";
   #_w3 := NOT #_w2 AND #"n_trig[28]";   // falling edge
   #"n_trig[28]" := #_w2;
   IF #_w3 THEN #"Step" := 23; END_IF;
   IF #_w1 THEN #lift := TRUE; END_IF;
END_REGION

REGION Network 17
   RUNG wire#powerrail
      Contact( #Unload_Sequence_Active )
      { S7_Templates := "SrcType := Int" } EQ_Contact(in1 := #"Step", in2 := 23)
      wire#w1
      Contact( #"at middle" )
      Move(in := 24, out1 => #"Step")
   END_RUNG
   RUNG wire#w1
      R_Coil( #forks_right )
   END_RUNG
   // the same network as SCL:
   #_w1 := #Unload_Sequence_Active AND (#"Step" = 23);
   IF #_w1 AND #"at middle" THEN #"Step" := 24; END_IF;
   IF #_w1 THEN #forks_right := FALSE; END_IF;
END_REGION

REGION Network 18
   RUNG wire#powerrail
      Contact( #Unload_Sequence_Active )
      { S7_Templates := "SrcType := Int" } EQ_Contact(in1 := #"Step", in2 := 24)
      wire#w1
      Contact( #"moving Z" )
      N_Trig( #"n_trig[29]" )
      Move(in := 25, out1 => #"Step")
   END_RUNG
   RUNG wire#w1
      R_Coil( #lift )
   END_RUNG
   // the same network as SCL:
   #_w1 := #Unload_Sequence_Active AND (#"Step" = 24);
   #_w2 := #_w1 AND #"moving Z";
   #_w3 := NOT #_w2 AND #"n_trig[29]";   // falling edge
   #"n_trig[29]" := #_w2;
   IF #_w3 THEN #"Step" := 25; END_IF;
   IF #_w1 THEN #lift := FALSE; END_IF;
END_REGION

REGION Network 19
   RUNG wire#powerrail
      Contact( #Unload_Sequence_Active )
      { S7_Templates := "SrcType := Int" } EQ_Contact(in1 := #"Step", in2 := 25)
      wire#w1
      Contact( #"moving X" )
      N_Trig( #"n_trig[30]" )
      Move(in := 26, out1 => #"Step")
   END_RUNG
   RUNG wire#w1
      Move(in := 100, out1 => #target_position)
      R_Coil( #lift )
   END_RUNG
   // the same network as SCL:
   #_w1 := #Unload_Sequence_Active AND (#"Step" = 25);
   #_w2 := #_w1 AND #"moving X";
   #_w3 := NOT #_w2 AND #"n_trig[30]";   // falling edge
   #"n_trig[30]" := #_w2;
   IF #_w3 THEN #"Step" := 26; END_IF;
   IF #_w1 THEN
       #target_position := 100;
       #lift := FALSE;
   END_IF;
END_REGION

REGION Network 20
   RUNG wire#powerrail
      Contact( #Unload_Sequence_Active )
      { S7_Templates := "SrcType := Int" } EQ_Contact(in1 := #"Step", in2 := 26)
      wire#w1
      Contact( #"moving Z" )
      N_Trig( #"n_trig[31]" )
      Move(in := 27, out1 => #"Step")
   END_RUNG
   RUNG wire#w1
      S_Coil( #lift )
   END_RUNG
   // the same network as SCL:
   #_w1 := #Unload_Sequence_Active AND (#"Step" = 26);
   #_w2 := #_w1 AND #"moving Z";
   #_w3 := NOT #_w2 AND #"n_trig[31]";   // falling edge
   #"n_trig[31]" := #_w2;
   IF #_w3 THEN #"Step" := 27; END_IF;
   IF #_w1 THEN #lift := TRUE; END_IF;
END_REGION

REGION Network 21
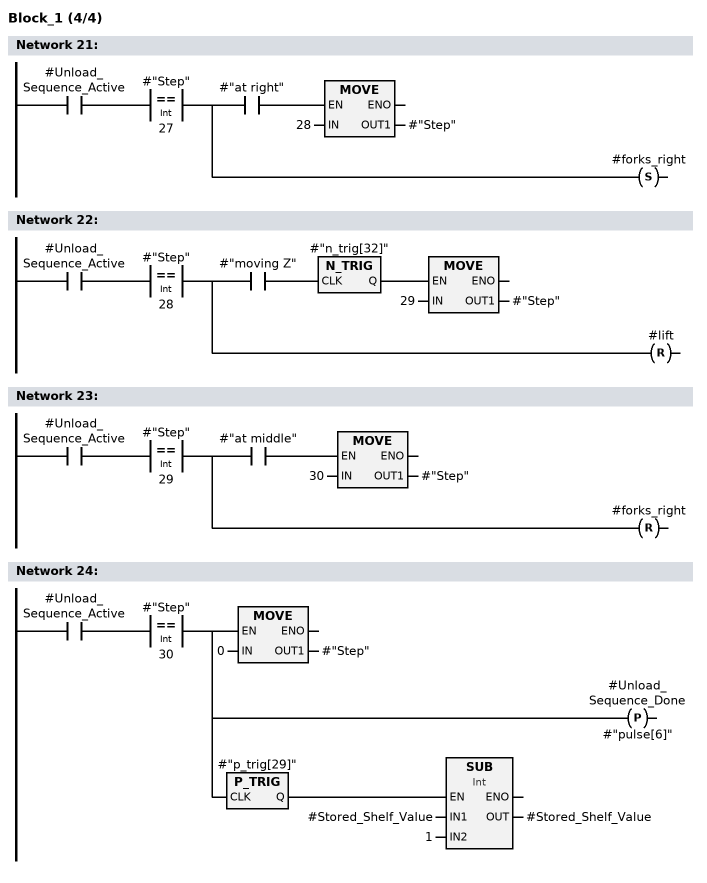
   RUNG wire#powerrail
      Contact( #Unload_Sequence_Active )
      { S7_Templates := "SrcType := Int" } EQ_Contact(in1 := #"Step", in2 := 27)
      wire#w1
      Contact( #"at right" )
      Move(in := 28, out1 => #"Step")
   END_RUNG
   RUNG wire#w1
      S_Coil( #forks_right )
   END_RUNG
   // the same network as SCL:
   #_w1 := #Unload_Sequence_Active AND (#"Step" = 27);
   IF #_w1 AND #"at right" THEN #"Step" := 28; END_IF;
   IF #_w1 THEN #forks_right := TRUE; END_IF;
END_REGION

REGION Network 22
   RUNG wire#powerrail
      Contact( #Unload_Sequence_Active )
      { S7_Templates := "SrcType := Int" } EQ_Contact(in1 := #"Step", in2 := 28)
      wire#w1
      Contact( #"moving Z" )
      N_Trig( #"n_trig[32]" )
      Move(in := 29, out1 => #"Step")
   END_RUNG
   RUNG wire#w1
      R_Coil( #lift )
   END_RUNG
   // the same network as SCL:
   #_w1 := #Unload_Sequence_Active AND (#"Step" = 28);
   #_w2 := #_w1 AND #"moving Z";
   #_w3 := NOT #_w2 AND #"n_trig[32]";   // falling edge
   #"n_trig[32]" := #_w2;
   IF #_w3 THEN #"Step" := 29; END_IF;
   IF #_w1 THEN #lift := FALSE; END_IF;
END_REGION

REGION Network 23
   RUNG wire#powerrail
      Contact( #Unload_Sequence_Active )
      { S7_Templates := "SrcType := Int" } EQ_Contact(in1 := #"Step", in2 := 29)
      wire#w1
      Contact( #"at middle" )
      Move(in := 30, out1 => #"Step")
   END_RUNG
   RUNG wire#w1
      R_Coil( #forks_right )
   END_RUNG
   // the same network as SCL:
   #_w1 := #Unload_Sequence_Active AND (#"Step" = 29);
   IF #_w1 AND #"at middle" THEN #"Step" := 30; END_IF;
   IF #_w1 THEN #forks_right := FALSE; END_IF;
END_REGION

REGION Network 24
   #_w1 := #Unload_Sequence_Active AND (#"Step" = 30);
   IF #_w1 THEN #"Step" := 0; END_IF;
   #Unload_Sequence_Done := #_w1 AND NOT #"pulse[6]";   // rising edge
   #"pulse[6]" := #_w1;
   #_w2 := #_w1 AND NOT #"p_trig[29]";   // rising edge
   #"p_trig[29]" := #_w1;
   IF #_w2 THEN #Stored_Shelf_Value := #Stored_Shelf_Value - 1; END_IF;
END_REGION
END_FUNCTION_BLOCK

FUNCTION_BLOCK "Block_2"   // FB6, LAD
{ S7_Optimized_Access := 'TRUE' }
VERSION : 0.1
   VAR_INPUT
      at_entry : Bool;
      at_load : Bool;
      at_unload : Bool;
      at_exit : Bool;
      shelf_value : Int;
   END_VAR
   VAR_OUTPUT
      entry_conveyor : Bool;
      load_conveyor : Bool;
      unload_conveyor : Bool;
      exit_conveyor : Bool;
   END_VAR
BEGIN

REGION Network 1
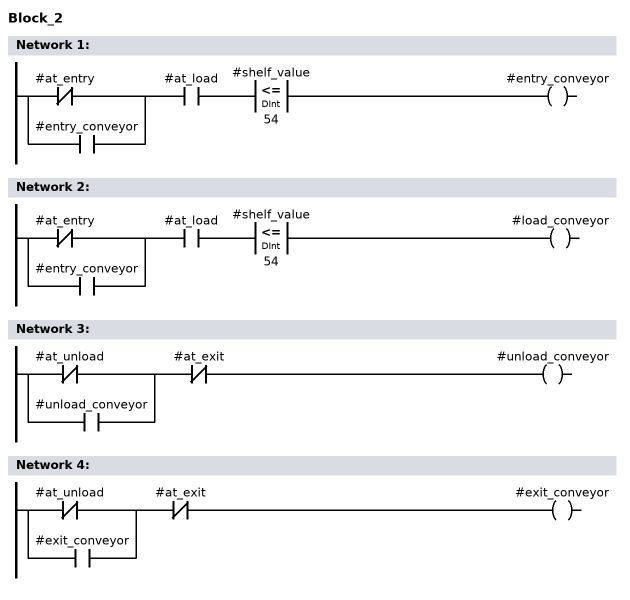
   RUNG wire#powerrail
      I_Contact( #at_entry )
      wire#w1
      Contact( #at_load )
      { S7_Templates := "SrcType := DInt" } LE_Contact(in1 := #shelf_value, in2 := 54)
      Coil( #entry_conveyor )
   END_RUNG
   RUNG wire#powerrail
      Contact( #entry_conveyor )
   END_RUNG wire#w1
   // the same network as SCL:
   #entry_conveyor := (NOT #at_entry OR #entry_conveyor) AND #at_load AND (#shelf_value <= 54);
END_REGION

REGION Network 2
   RUNG wire#powerrail
      I_Contact( #at_entry )
      wire#w1
      Contact( #at_load )
      { S7_Templates := "SrcType := DInt" } LE_Contact(in1 := #shelf_value, in2 := 54)
      Coil( #load_conveyor )
   END_RUNG
   RUNG wire#powerrail
      Contact( #entry_conveyor )
   END_RUNG wire#w1
   // the same network as SCL:
   #load_conveyor := (NOT #at_entry OR #entry_conveyor) AND #at_load AND (#shelf_value <= 54);
END_REGION

REGION Network 3
   RUNG wire#powerrail
      I_Contact( #at_unload )
      wire#w1
      I_Contact( #at_exit )
      Coil( #unload_conveyor )
   END_RUNG
   RUNG wire#powerrail
      Contact( #unload_conveyor )
   END_RUNG wire#w1
   // the same network as SCL:
   #unload_conveyor := (NOT #at_unload OR #unload_conveyor) AND NOT #at_exit;
END_REGION

REGION Network 4
   RUNG wire#powerrail
      I_Contact( #at_unload )
      wire#w1
      I_Contact( #at_exit )
      Coil( #exit_conveyor )
   END_RUNG
   RUNG wire#powerrail
      Contact( #exit_conveyor )
   END_RUNG wire#w1
   // the same network as SCL:
   #exit_conveyor := (NOT #at_unload OR #exit_conveyor) AND NOT #at_exit;
END_REGION
END_FUNCTION_BLOCK

FUNCTION "MHJ-PLC-Lab-Function-S71200" : Void   // FC9000, SCL
{ S7_Optimized_Access := 'TRUE' }
VERSION : 0.1
   VAR_TEMP
      rdTimeReturn : Int;
      outputTime : DTL;
      SyncVal : Byte;
      forVal : Int;
      forVal_2 : Int;
      Value : Byte;
   END_VAR
   VAR CONSTANT
      CompVal : Byte := 16#34;
      Value_01 : Byte := 16#11;
      Value_01_DW : DWord := 16#A165_D992;
      Value_02_DW : DWord := 16#58BE_4401;
   END_VAR
BEGIN

   #Value:=PEEK(area := 16#82,
        dbNumber := 0,
        byteOffset := 511);
   #Value := #Value + 1;

   POKE(area := 16#82,
        dbNumber := 0,
        byteOffset := 511,
        value := #Value);

   POKE(area:=16#81,
        dbNumber:=0,
        byteOffset:=1016,
        value:=#Value_01_DW);
   POKE(area := 16#81,
        dbNumber := 0,
        byteOffset := 1020,
        value := #Value_02_DW);

   POKE(area := 16#81,
        dbNumber := 0,
        byteOffset := 511,
        value := B#16#00);

   FOR #forVal := 0 TO 120 DO
       FOR #forVal_2:=0 TO 10 DO
           #rdTimeReturn:=RD_SYS_T(#outputTime);
           #rdTimeReturn := WR_SYS_T(#outputTime);
           #rdTimeReturn := RD_SYS_T(#outputTime);
           #rdTimeReturn := WR_SYS_T(#outputTime);
       END_FOR;
       #SyncVal:= PEEK(area := 16#81,
                      dbNumber := 0,
                      byteOffset := 511);
       IF #SyncVal = #CompVal THEN
          GOTO M_1;
       END_IF;
   END_FOR;
   RETURN;

   M_1:
   POKE(area := 16#81,
        dbNumber := 0,
        byteOffset := 511,
        value := B#16#0);
END_FUNCTION

ORGANIZATION_BLOCK "Main"   // OB1, LAD, ProgramCycle
TITLE = "Main Program Sweep (Cycle)"
{ S7_Optimized_Access := 'TRUE' }
VERSION : 0.1
   VAR_INPUT
      Initial_Call : Bool;   // Initial call of this OB
      Remanence : Bool;   // =True, if remanent data are available
   END_VAR
   VAR_TEMP   // added for the SCL form of the ladder/FBD networks
      _w1 : Bool;
      _w2 : Bool;
      _w3 : Bool;
      _w4 : Bool;
   END_VAR
BEGIN

REGION Network 1: Konnektierungsbaustein für PLC-Lab
   // Im Netzwerk 1 wird der Konnektierungsbaustein für PLC-Lab aufgerufen.
   // Dieser Aufruf darf nicht entfernt werden!
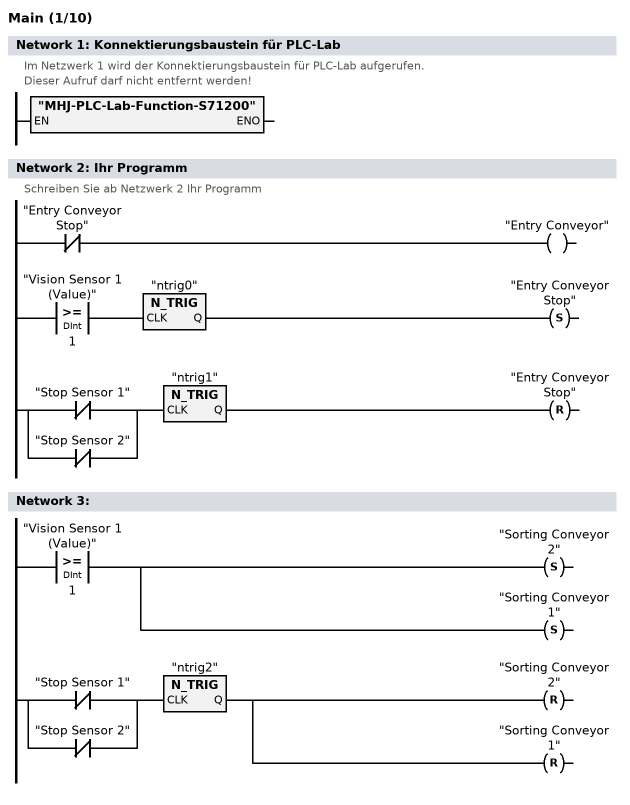
   RUNG wire#powerrail
      "MHJ-PLC-Lab-Function-S71200"()
   END_RUNG
   // the same network as SCL:
   "MHJ-PLC-Lab-Function-S71200"();
END_REGION

REGION Network 2: Ihr Programm
   // Schreiben Sie ab Netzwerk 2 Ihr Programm
   RUNG wire#powerrail
      I_Contact( "Entry Conveyor Stop" )
      Coil( "Entry Conveyor" )
   END_RUNG
   RUNG wire#powerrail
      { S7_Templates := "SrcType := DInt" } GE_Contact(in1 := "Vision Sensor 1 (Value)", in2 := 1)
      N_Trig( "ntrig0" )
      S_Coil( "Entry Conveyor Stop" )
   END_RUNG
   RUNG wire#powerrail
      I_Contact( "Stop Sensor 1" )
      wire#w1
      N_Trig( "ntrig1" )
      R_Coil( "Entry Conveyor Stop" )
   END_RUNG
   RUNG wire#powerrail
      I_Contact( "Stop Sensor 2" )
   END_RUNG wire#w1
   // the same network as SCL:
   "Entry Conveyor" := NOT "Entry Conveyor Stop";
   #_w1 := "Vision Sensor 1 (Value)" >= 1;
   #_w2 := NOT #_w1 AND "ntrig0";   // falling edge
   "ntrig0" := #_w1;
   IF #_w2 THEN "Entry Conveyor Stop" := TRUE; END_IF;
   #_w3 := NOT "Stop Sensor 1" OR NOT "Stop Sensor 2";
   #_w4 := NOT #_w3 AND "ntrig1";   // falling edge
   "ntrig1" := #_w3;
   IF #_w4 THEN "Entry Conveyor Stop" := FALSE; END_IF;
END_REGION

REGION Network 3
   RUNG wire#powerrail
      { S7_Templates := "SrcType := DInt" } GE_Contact(in1 := "Vision Sensor 1 (Value)", in2 := 1)
      wire#w1
      S_Coil( "Sorting Conveyor 2" )
   END_RUNG
   RUNG wire#w1
      S_Coil( "Sorting Conveyor 1" )
   END_RUNG
   RUNG wire#powerrail
      I_Contact( "Stop Sensor 1" )
      wire#w2
      N_Trig( "ntrig2" )
      wire#w3
      R_Coil( "Sorting Conveyor 2" )
   END_RUNG
   RUNG wire#powerrail
      I_Contact( "Stop Sensor 2" )
   END_RUNG wire#w2
   RUNG wire#w3
      R_Coil( "Sorting Conveyor 1" )
   END_RUNG
   // the same network as SCL:
   IF "Vision Sensor 1 (Value)" >= 1 THEN
       "Sorting Conveyor 2" := TRUE;
       "Sorting Conveyor 1" := TRUE;
   END_IF;
   #_w1 := NOT "Stop Sensor 1" OR NOT "Stop Sensor 2";
   #_w2 := NOT #_w1 AND "ntrig2";   // falling edge
   "ntrig2" := #_w1;
   IF #_w2 THEN
       "Sorting Conveyor 2" := FALSE;
       "Sorting Conveyor 1" := FALSE;
   END_IF;
END_REGION

REGION Network 4: Vision Sensor Database
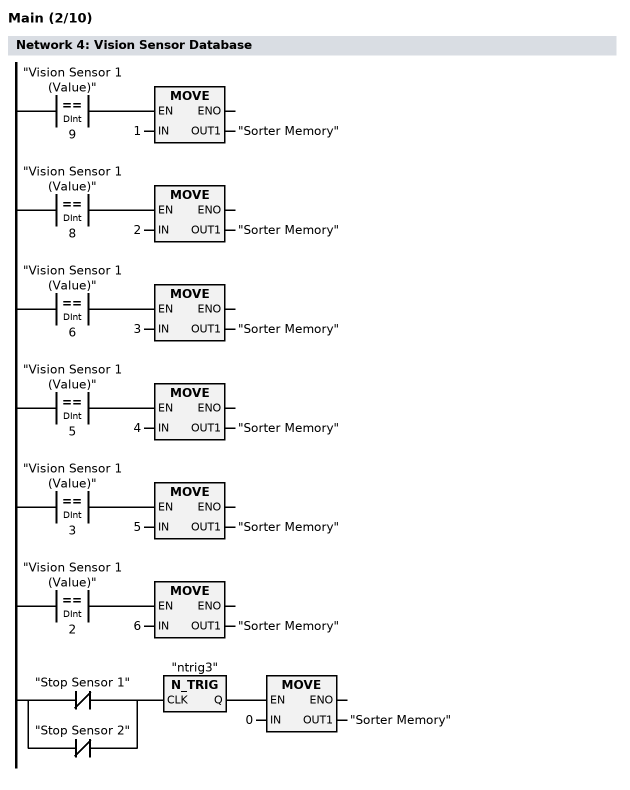
   RUNG wire#powerrail
      { S7_Templates := "SrcType := DInt" } EQ_Contact(in1 := "Vision Sensor 1 (Value)", in2 := 9)
      Move(in := 1, out1 => "Sorter Memory")
   END_RUNG
   RUNG wire#powerrail
      { S7_Templates := "SrcType := DInt" } EQ_Contact(in1 := "Vision Sensor 1 (Value)", in2 := 8)
      Move(in := 2, out1 => "Sorter Memory")
   END_RUNG
   RUNG wire#powerrail
      { S7_Templates := "SrcType := DInt" } EQ_Contact(in1 := "Vision Sensor 1 (Value)", in2 := 6)
      Move(in := 3, out1 => "Sorter Memory")
   END_RUNG
   RUNG wire#powerrail
      { S7_Templates := "SrcType := DInt" } EQ_Contact(in1 := "Vision Sensor 1 (Value)", in2 := 5)
      Move(in := 4, out1 => "Sorter Memory")
   END_RUNG
   RUNG wire#powerrail
      { S7_Templates := "SrcType := DInt" } EQ_Contact(in1 := "Vision Sensor 1 (Value)", in2 := 3)
      Move(in := 5, out1 => "Sorter Memory")
   END_RUNG
   RUNG wire#powerrail
      { S7_Templates := "SrcType := DInt" } EQ_Contact(in1 := "Vision Sensor 1 (Value)", in2 := 2)
      Move(in := 6, out1 => "Sorter Memory")
   END_RUNG
   RUNG wire#powerrail
      I_Contact( "Stop Sensor 1" )
      wire#w1
      N_Trig( "ntrig3" )
      Move(in := 0, out1 => "Sorter Memory")
   END_RUNG
   RUNG wire#powerrail
      I_Contact( "Stop Sensor 2" )
   END_RUNG wire#w1
   // the same network as SCL:
   IF "Vision Sensor 1 (Value)" = 9 THEN "Sorter Memory" := 1; END_IF;
   IF "Vision Sensor 1 (Value)" = 8 THEN "Sorter Memory" := 2; END_IF;
   IF "Vision Sensor 1 (Value)" = 6 THEN "Sorter Memory" := 3; END_IF;
   IF "Vision Sensor 1 (Value)" = 5 THEN "Sorter Memory" := 4; END_IF;
   IF "Vision Sensor 1 (Value)" = 3 THEN "Sorter Memory" := 5; END_IF;
   IF "Vision Sensor 1 (Value)" = 2 THEN "Sorter Memory" := 6; END_IF;
   #_w1 := NOT "Stop Sensor 1" OR NOT "Stop Sensor 2";
   #_w2 := NOT #_w1 AND "ntrig3";   // falling edge
   "ntrig3" := #_w1;
   IF #_w2 THEN "Sorter Memory" := 0; END_IF;
END_REGION

REGION Network 5: Sorting Arms Database
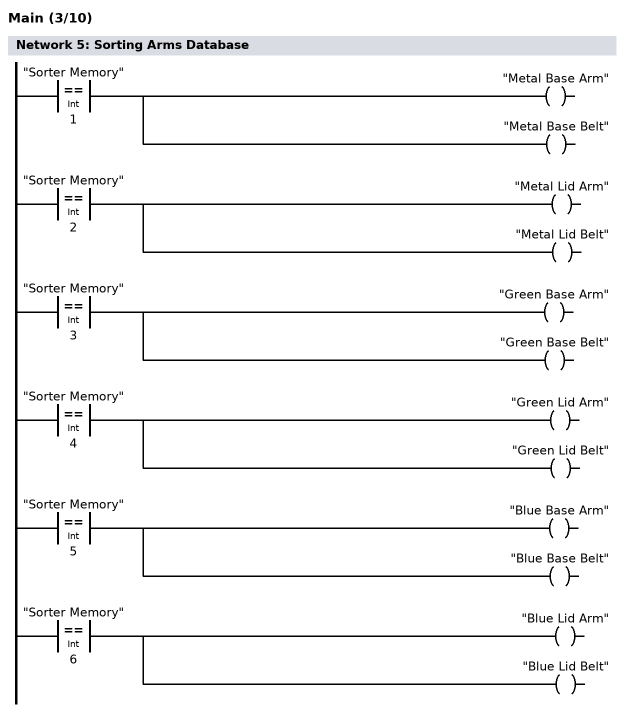
   RUNG wire#powerrail
      { S7_Templates := "SrcType := Int" } EQ_Contact(in1 := "Sorter Memory", in2 := 1)
      wire#w1
      Coil( "Metal Base Arm" )
   END_RUNG
   RUNG wire#w1
      Coil( "Metal Base Belt" )
   END_RUNG
   RUNG wire#powerrail
      { S7_Templates := "SrcType := Int" } EQ_Contact(in1 := "Sorter Memory", in2 := 2)
      wire#w2
      Coil( "Metal Lid Arm" )
   END_RUNG
   RUNG wire#w2
      Coil( "Metal Lid Belt" )
   END_RUNG
   RUNG wire#powerrail
      { S7_Templates := "SrcType := Int" } EQ_Contact(in1 := "Sorter Memory", in2 := 3)
      wire#w3
      Coil( "Green Base Arm" )
   END_RUNG
   RUNG wire#w3
      Coil( "Green Base Belt" )
   END_RUNG
   RUNG wire#powerrail
      { S7_Templates := "SrcType := Int" } EQ_Contact(in1 := "Sorter Memory", in2 := 4)
      wire#w4
      Coil( "Green Lid Arm" )
   END_RUNG
   RUNG wire#w4
      Coil( "Green Lid Belt" )
   END_RUNG
   RUNG wire#powerrail
      { S7_Templates := "SrcType := Int" } EQ_Contact(in1 := "Sorter Memory", in2 := 5)
      wire#w5
      Coil( "Blue Base Arm" )
   END_RUNG
   RUNG wire#w5
      Coil( "Blue Base Belt" )
   END_RUNG
   RUNG wire#powerrail
      { S7_Templates := "SrcType := Int" } EQ_Contact(in1 := "Sorter Memory", in2 := 6)
      wire#w6
      Coil( "Blue Lid Arm" )
   END_RUNG
   RUNG wire#w6
      Coil( "Blue Lid Belt" )
   END_RUNG
   // the same network as SCL:
   "Metal Base Arm" := "Sorter Memory" = 1;
   "Metal Base Belt" := "Metal Base Arm";
   "Metal Lid Arm" := "Sorter Memory" = 2;
   "Metal Lid Belt" := "Metal Lid Arm";
   "Green Base Arm" := "Sorter Memory" = 3;
   "Green Base Belt" := "Green Base Arm";
   "Green Lid Arm" := "Sorter Memory" = 4;
   "Green Lid Belt" := "Green Lid Arm";
   "Blue Base Arm" := "Sorter Memory" = 5;
   "Blue Base Belt" := "Blue Base Arm";
   "Blue Lid Arm" := "Sorter Memory" = 6;
   "Blue Lid Belt" := "Blue Lid Arm";
END_REGION

REGION Network 6: Base Clamp Conveyors
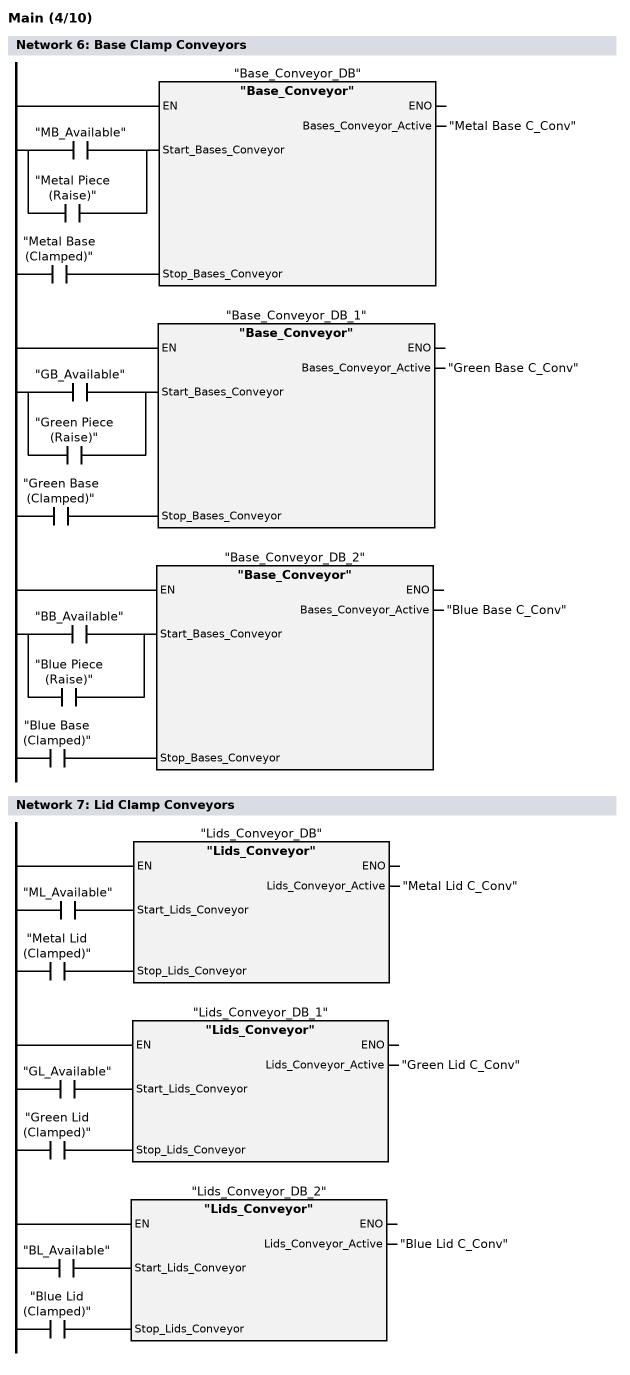
   RUNG wire#powerrail
      "Base_Conveyor_DB"(Start_Bases_Conveyor := wire#w1, Stop_Bases_Conveyor := wire#w2, Bases_Conveyor_Active => "Metal Base C_Conv")
   END_RUNG
   RUNG wire#powerrail
      Contact( "MB_Available" )
   END_RUNG wire#w1
   RUNG wire#powerrail
      Contact( "Metal Piece (Raise)" )
   END_RUNG wire#w1
   RUNG wire#powerrail
      Contact( "Metal Base (Clamped)" )
   END_RUNG wire#w2
   RUNG wire#powerrail
      "Base_Conveyor_DB_1"(Start_Bases_Conveyor := wire#w3, Stop_Bases_Conveyor := wire#w4, Bases_Conveyor_Active => "Green Base C_Conv")
   END_RUNG
   RUNG wire#powerrail
      Contact( "GB_Available" )
   END_RUNG wire#w3
   RUNG wire#powerrail
      Contact( "Green Piece (Raise)" )
   END_RUNG wire#w3
   RUNG wire#powerrail
      Contact( "Green Base (Clamped)" )
   END_RUNG wire#w4
   RUNG wire#powerrail
      "Base_Conveyor_DB_2"(Start_Bases_Conveyor := wire#w5, Stop_Bases_Conveyor := wire#w6, Bases_Conveyor_Active => "Blue Base C_Conv")
   END_RUNG
   RUNG wire#powerrail
      Contact( "BB_Available" )
   END_RUNG wire#w5
   RUNG wire#powerrail
      Contact( "Blue Piece (Raise)" )
   END_RUNG wire#w5
   RUNG wire#powerrail
      Contact( "Blue Base (Clamped)" )
   END_RUNG wire#w6
   // the same network as SCL:
   "Base_Conveyor_DB"(Start_Bases_Conveyor := "MB_Available" OR "Metal Piece (Raise)",   // "Base_Conveyor"
                      Stop_Bases_Conveyor := "Metal Base (Clamped)",
                      Bases_Conveyor_Active => "Metal Base C_Conv");
   "Base_Conveyor_DB_1"(Start_Bases_Conveyor := "GB_Available" OR "Green Piece (Raise)",   // "Base_Conveyor"
                        Stop_Bases_Conveyor := "Green Base (Clamped)",
                        Bases_Conveyor_Active => "Green Base C_Conv");
   "Base_Conveyor_DB_2"(Start_Bases_Conveyor := "BB_Available" OR "Blue Piece (Raise)",   // "Base_Conveyor"
                        Stop_Bases_Conveyor := "Blue Base (Clamped)",
                        Bases_Conveyor_Active => "Blue Base C_Conv");
END_REGION

REGION Network 7: Lid Clamp Conveyors
   RUNG wire#powerrail
      "Lids_Conveyor_DB"(Start_Lids_Conveyor := wire#w1, Stop_Lids_Conveyor := wire#w2, Lids_Conveyor_Active => "Metal Lid C_Conv")
   END_RUNG
   RUNG wire#powerrail
      Contact( "ML_Available" )
   END_RUNG wire#w1
   RUNG wire#powerrail
      Contact( "Metal Lid (Clamped)" )
   END_RUNG wire#w2
   RUNG wire#powerrail
      "Lids_Conveyor_DB_1"(Start_Lids_Conveyor := wire#w3, Stop_Lids_Conveyor := wire#w4, Lids_Conveyor_Active => "Green Lid C_Conv")
   END_RUNG
   RUNG wire#powerrail
      Contact( "GL_Available" )
   END_RUNG wire#w3
   RUNG wire#powerrail
      Contact( "Green Lid (Clamped)" )
   END_RUNG wire#w4
   RUNG wire#powerrail
      "Lids_Conveyor_DB_2"(Start_Lids_Conveyor := wire#w5, Stop_Lids_Conveyor := wire#w6, Lids_Conveyor_Active => "Blue Lid C_Conv")
   END_RUNG
   RUNG wire#powerrail
      Contact( "BL_Available" )
   END_RUNG wire#w5
   RUNG wire#powerrail
      Contact( "Blue Lid (Clamped)" )
   END_RUNG wire#w6
   // the same network as SCL:
   "Lids_Conveyor_DB"(Start_Lids_Conveyor := "ML_Available",   // "Lids_Conveyor"
                      Stop_Lids_Conveyor := "Metal Lid (Clamped)",
                      Lids_Conveyor_Active => "Metal Lid C_Conv");
   "Lids_Conveyor_DB_1"(Start_Lids_Conveyor := "GL_Available",   // "Lids_Conveyor"
                        Stop_Lids_Conveyor := "Green Lid (Clamped)",
                        Lids_Conveyor_Active => "Green Lid C_Conv");
   "Lids_Conveyor_DB_2"(Start_Lids_Conveyor := "BL_Available",   // "Lids_Conveyor"
                        Stop_Lids_Conveyor := "Blue Lid (Clamped)",
                        Lids_Conveyor_Active => "Blue Lid C_Conv");
END_REGION

REGION Network 8: Clamping Blocks
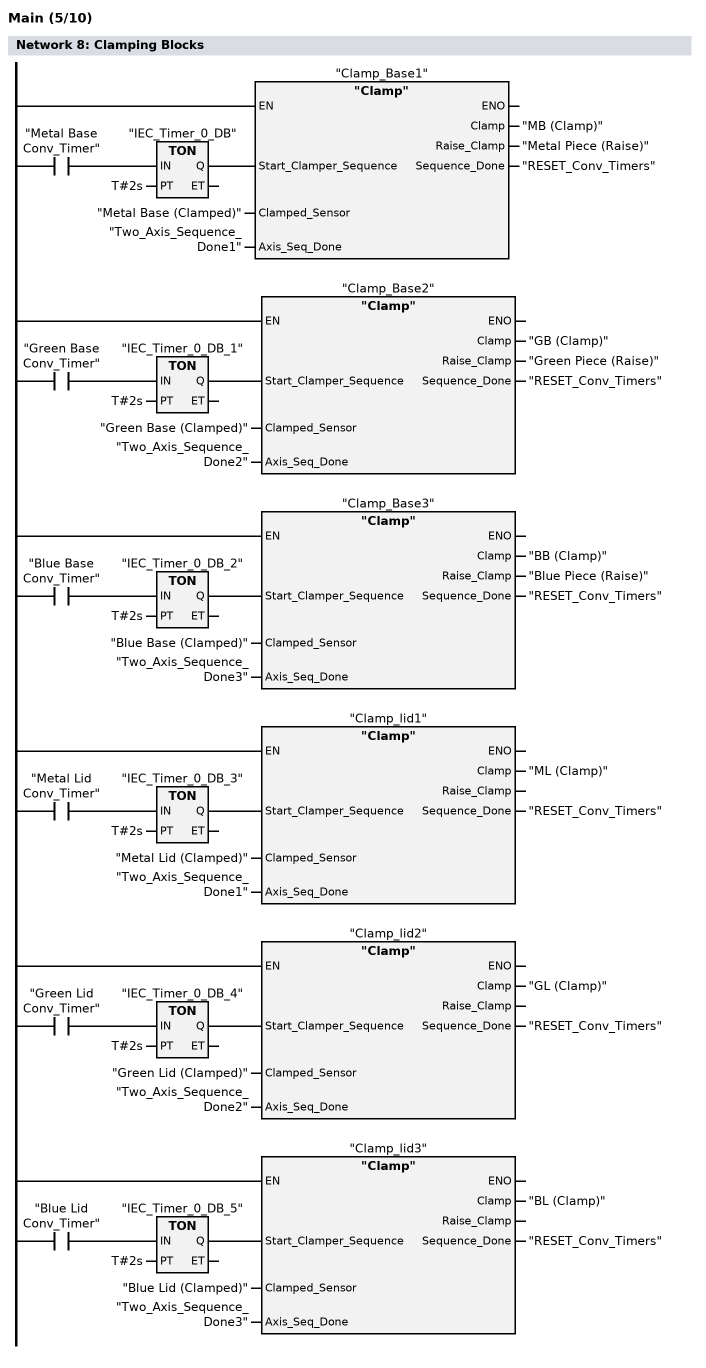
   "IEC_Timer_0_DB".TON(IN := "Metal Base Conv_Timer", PT := T#2s);
   "Clamp_Base1"(Start_Clamper_Sequence := "IEC_Timer_0_DB".Q,   // "Clamp"
                 Clamped_Sensor := "Metal Base (Clamped)",
                 Axis_Seq_Done := "Two_Axis_Sequence_Done1",
                 Clamp => "MB (Clamp)",
                 Raise_Clamp => "Metal Piece (Raise)",
                 Sequence_Done => "RESET_Conv_Timers");
   "IEC_Timer_0_DB_1".TON(IN := "Green Base Conv_Timer", PT := T#2s);
   "Clamp_Base2"(Start_Clamper_Sequence := "IEC_Timer_0_DB_1".Q,   // "Clamp"
                 Clamped_Sensor := "Green Base (Clamped)",
                 Axis_Seq_Done := "Two_Axis_Sequence_Done2",
                 Clamp => "GB (Clamp)",
                 Raise_Clamp => "Green Piece (Raise)",
                 Sequence_Done => "RESET_Conv_Timers");
   "IEC_Timer_0_DB_2".TON(IN := "Blue Base Conv_Timer", PT := T#2s);
   "Clamp_Base3"(Start_Clamper_Sequence := "IEC_Timer_0_DB_2".Q,   // "Clamp"
                 Clamped_Sensor := "Blue Base (Clamped)",
                 Axis_Seq_Done := "Two_Axis_Sequence_Done3",
                 Clamp => "BB (Clamp)",
                 Raise_Clamp => "Blue Piece (Raise)",
                 Sequence_Done => "RESET_Conv_Timers");
   "IEC_Timer_0_DB_3".TON(IN := "Metal Lid Conv_Timer", PT := T#2s);
   "Clamp_lid1"(Start_Clamper_Sequence := "IEC_Timer_0_DB_3".Q,   // "Clamp"
                Clamped_Sensor := "Metal Lid (Clamped)",
                Axis_Seq_Done := "Two_Axis_Sequence_Done1",
                Clamp => "ML (Clamp)",
                Sequence_Done => "RESET_Conv_Timers");
   "IEC_Timer_0_DB_4".TON(IN := "Green Lid Conv_Timer", PT := T#2s);
   "Clamp_lid2"(Start_Clamper_Sequence := "IEC_Timer_0_DB_4".Q,   // "Clamp"
                Clamped_Sensor := "Green Lid (Clamped)",
                Axis_Seq_Done := "Two_Axis_Sequence_Done2",
                Clamp => "GL (Clamp)",
                Sequence_Done => "RESET_Conv_Timers");
   "IEC_Timer_0_DB_5".TON(IN := "Blue Lid Conv_Timer", PT := T#2s);
   "Clamp_lid3"(Start_Clamper_Sequence := "IEC_Timer_0_DB_5".Q,   // "Clamp"
                Clamped_Sensor := "Blue Lid (Clamped)",
                Axis_Seq_Done := "Two_Axis_Sequence_Done3",
                Clamp => "BL (Clamp)",
                Sequence_Done => "RESET_Conv_Timers");
END_REGION

REGION Network 9: Clamping latches setters
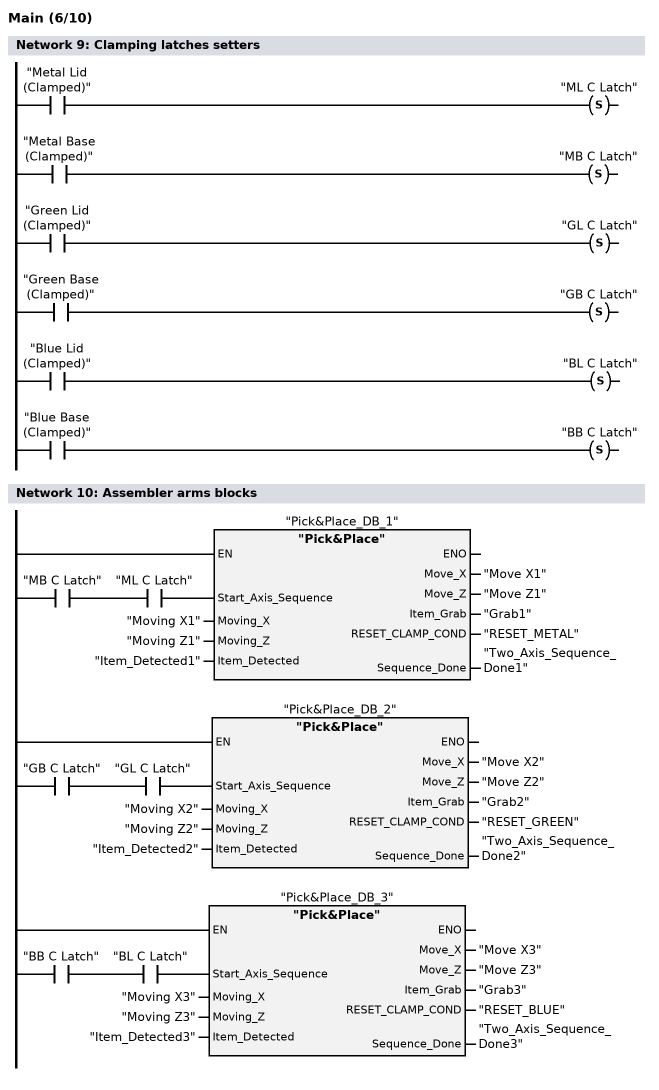
   RUNG wire#powerrail
      Contact( "Metal Lid (Clamped)" )
      S_Coil( "ML C Latch" )
   END_RUNG
   RUNG wire#powerrail
      Contact( "Metal Base (Clamped)" )
      S_Coil( "MB C Latch" )
   END_RUNG
   RUNG wire#powerrail
      Contact( "Green Lid (Clamped)" )
      S_Coil( "GL C Latch" )
   END_RUNG
   RUNG wire#powerrail
      Contact( "Green Base (Clamped)" )
      S_Coil( "GB C Latch" )
   END_RUNG
   RUNG wire#powerrail
      Contact( "Blue Lid (Clamped)" )
      S_Coil( "BL C Latch" )
   END_RUNG
   RUNG wire#powerrail
      Contact( "Blue Base (Clamped)" )
      S_Coil( "BB C Latch" )
   END_RUNG
   // the same network as SCL:
   IF "Metal Lid (Clamped)" THEN "ML C Latch" := TRUE; END_IF;
   IF "Metal Base (Clamped)" THEN "MB C Latch" := TRUE; END_IF;
   IF "Green Lid (Clamped)" THEN "GL C Latch" := TRUE; END_IF;
   IF "Green Base (Clamped)" THEN "GB C Latch" := TRUE; END_IF;
   IF "Blue Lid (Clamped)" THEN "BL C Latch" := TRUE; END_IF;
   IF "Blue Base (Clamped)" THEN "BB C Latch" := TRUE; END_IF;
END_REGION

REGION Network 10: Assembler arms blocks
   RUNG wire#powerrail
      "Pick&Place_DB_1"(Start_Axis_Sequence := wire#w1, Moving_X := "Moving X1", Moving_Z := "Moving Z1", Item_Detected := "Item_Detected1", Move_X => "Move X1", Move_Z => "Move Z1", Item_Grab => "Grab1", RESET_CLAMP_COND => "RESET_METAL", Sequence_Done => "Two_Axis_Sequence_Done1")
   END_RUNG
   RUNG wire#powerrail
      Contact( "MB C Latch" )
      Contact( "ML C Latch" )
   END_RUNG wire#w1
   RUNG wire#powerrail
      "Pick&Place_DB_2"(Start_Axis_Sequence := wire#w2, Moving_X := "Moving X2", Moving_Z := "Moving Z2", Item_Detected := "Item_Detected2", Move_X => "Move X2", Move_Z => "Move Z2", Item_Grab => "Grab2", RESET_CLAMP_COND => "RESET_GREEN", Sequence_Done => "Two_Axis_Sequence_Done2")
   END_RUNG
   RUNG wire#powerrail
      Contact( "GB C Latch" )
      Contact( "GL C Latch" )
   END_RUNG wire#w2
   RUNG wire#powerrail
      "Pick&Place_DB_3"(Start_Axis_Sequence := wire#w3, Moving_X := "Moving X3", Moving_Z := "Moving Z3", Item_Detected := "Item_Detected3", Move_X => "Move X3", Move_Z => "Move Z3", Item_Grab => "Grab3", RESET_CLAMP_COND => "RESET_BLUE", Sequence_Done => "Two_Axis_Sequence_Done3")
   END_RUNG
   RUNG wire#powerrail
      Contact( "BB C Latch" )
      Contact( "BL C Latch" )
   END_RUNG wire#w3
   // the same network as SCL:
   "Pick&Place_DB_1"(Start_Axis_Sequence := "MB C Latch" AND "ML C Latch",   // "Pick&Place"
                     Moving_X := "Moving X1",
                     Moving_Z := "Moving Z1",
                     Item_Detected := "Item_Detected1",
                     Move_X => "Move X1",
                     Move_Z => "Move Z1",
                     Item_Grab => "Grab1",
                     RESET_CLAMP_COND => "RESET_METAL",
                     Sequence_Done => "Two_Axis_Sequence_Done1");
   "Pick&Place_DB_2"(Start_Axis_Sequence := "GB C Latch" AND "GL C Latch",   // "Pick&Place"
                     Moving_X := "Moving X2",
                     Moving_Z := "Moving Z2",
                     Item_Detected := "Item_Detected2",
                     Move_X => "Move X2",
                     Move_Z => "Move Z2",
                     Item_Grab => "Grab2",
                     RESET_CLAMP_COND => "RESET_GREEN",
                     Sequence_Done => "Two_Axis_Sequence_Done2");
   "Pick&Place_DB_3"(Start_Axis_Sequence := "BB C Latch" AND "BL C Latch",   // "Pick&Place"
                     Moving_X := "Moving X3",
                     Moving_Z := "Moving Z3",
                     Item_Detected := "Item_Detected3",
                     Move_X => "Move X3",
                     Move_Z => "Move Z3",
                     Item_Grab => "Grab3",
                     RESET_CLAMP_COND => "RESET_BLUE",
                     Sequence_Done => "Two_Axis_Sequence_Done3");
END_REGION

REGION Network 11: Metal/Green/Blue latches resters
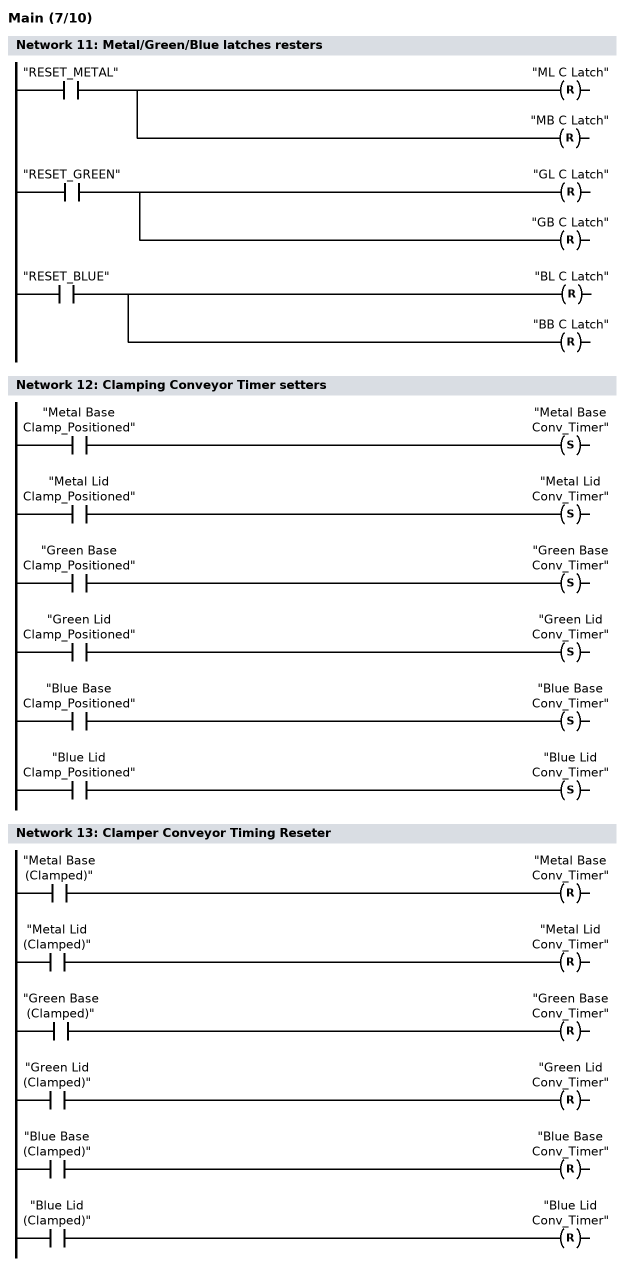
   RUNG wire#powerrail
      Contact( "RESET_METAL" )
      wire#w1
      R_Coil( "ML C Latch" )
   END_RUNG
   RUNG wire#w1
      R_Coil( "MB C Latch" )
   END_RUNG
   RUNG wire#powerrail
      Contact( "RESET_GREEN" )
      wire#w2
      R_Coil( "GL C Latch" )
   END_RUNG
   RUNG wire#w2
      R_Coil( "GB C Latch" )
   END_RUNG
   RUNG wire#powerrail
      Contact( "RESET_BLUE" )
      wire#w3
      R_Coil( "BL C Latch" )
   END_RUNG
   RUNG wire#w3
      R_Coil( "BB C Latch" )
   END_RUNG
   // the same network as SCL:
   IF "RESET_METAL" THEN
       "ML C Latch" := FALSE;
       "MB C Latch" := FALSE;
   END_IF;
   IF "RESET_GREEN" THEN
       "GL C Latch" := FALSE;
       "GB C Latch" := FALSE;
   END_IF;
   IF "RESET_BLUE" THEN
       "BL C Latch" := FALSE;
       "BB C Latch" := FALSE;
   END_IF;
END_REGION

REGION Network 12: Clamping Conveyor Timer setters
   RUNG wire#powerrail
      Contact( "Metal Base Clamp_Positioned" )
      S_Coil( "Metal Base Conv_Timer" )
   END_RUNG
   RUNG wire#powerrail
      Contact( "Metal Lid Clamp_Positioned" )
      S_Coil( "Metal Lid Conv_Timer" )
   END_RUNG
   RUNG wire#powerrail
      Contact( "Green Base Clamp_Positioned" )
      S_Coil( "Green Base Conv_Timer" )
   END_RUNG
   RUNG wire#powerrail
      Contact( "Green Lid Clamp_Positioned" )
      S_Coil( "Green Lid Conv_Timer" )
   END_RUNG
   RUNG wire#powerrail
      Contact( "Blue Base Clamp_Positioned" )
      S_Coil( "Blue Base Conv_Timer" )
   END_RUNG
   RUNG wire#powerrail
      Contact( "Blue Lid Clamp_Positioned" )
      S_Coil( "Blue Lid Conv_Timer" )
   END_RUNG
   // the same network as SCL:
   IF "Metal Base Clamp_Positioned" THEN "Metal Base Conv_Timer" := TRUE; END_IF;
   IF "Metal Lid Clamp_Positioned" THEN "Metal Lid Conv_Timer" := TRUE; END_IF;
   IF "Green Base Clamp_Positioned" THEN "Green Base Conv_Timer" := TRUE; END_IF;
   IF "Green Lid Clamp_Positioned" THEN "Green Lid Conv_Timer" := TRUE; END_IF;
   IF "Blue Base Clamp_Positioned" THEN "Blue Base Conv_Timer" := TRUE; END_IF;
   IF "Blue Lid Clamp_Positioned" THEN "Blue Lid Conv_Timer" := TRUE; END_IF;
END_REGION

REGION Network 13: Clamper Conveyor Timing Reseter
   RUNG wire#powerrail
      Contact( "Metal Base (Clamped)" )
      R_Coil( "Metal Base Conv_Timer" )
   END_RUNG
   RUNG wire#powerrail
      Contact( "Metal Lid (Clamped)" )
      R_Coil( "Metal Lid Conv_Timer" )
   END_RUNG
   RUNG wire#powerrail
      Contact( "Green Base (Clamped)" )
      R_Coil( "Green Base Conv_Timer" )
   END_RUNG
   RUNG wire#powerrail
      Contact( "Green Lid (Clamped)" )
      R_Coil( "Green Lid Conv_Timer" )
   END_RUNG
   RUNG wire#powerrail
      Contact( "Blue Base (Clamped)" )
      R_Coil( "Blue Base Conv_Timer" )
   END_RUNG
   RUNG wire#powerrail
      Contact( "Blue Lid (Clamped)" )
      R_Coil( "Blue Lid Conv_Timer" )
   END_RUNG
   // the same network as SCL:
   IF "Metal Base (Clamped)" THEN "Metal Base Conv_Timer" := FALSE; END_IF;
   IF "Metal Lid (Clamped)" THEN "Metal Lid Conv_Timer" := FALSE; END_IF;
   IF "Green Base (Clamped)" THEN "Green Base Conv_Timer" := FALSE; END_IF;
   IF "Green Lid (Clamped)" THEN "Green Lid Conv_Timer" := FALSE; END_IF;
   IF "Blue Base (Clamped)" THEN "Blue Base Conv_Timer" := FALSE; END_IF;
   IF "Blue Lid (Clamped)" THEN "Blue Lid Conv_Timer" := FALSE; END_IF;
END_REGION

REGION Network 14: Emitter Part Counter
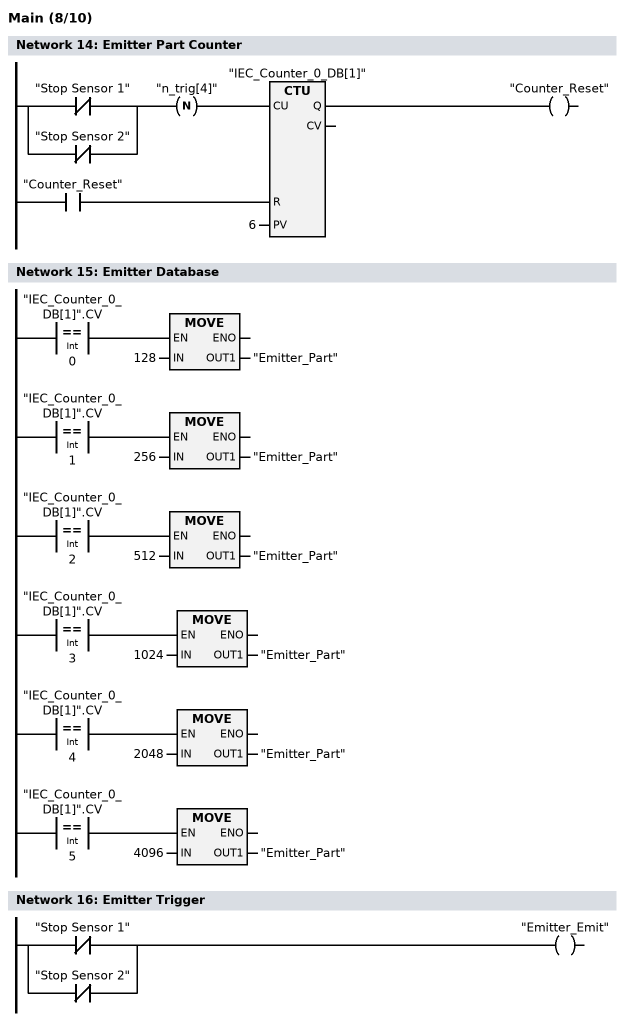
   #_w1 := NOT "Stop Sensor 1" OR NOT "Stop Sensor 2";
   #_w2 := NOT #_w1 AND "n_trig[4]";   // falling edge
   "n_trig[4]" := #_w1;
   "IEC_Counter_0_DB[1]".CTU(CU := #_w2, R := "Counter_Reset", PV := 6);
   "Counter_Reset" := "IEC_Counter_0_DB[1]".Q;
END_REGION

REGION Network 15: Emitter Database
   RUNG wire#powerrail
      { S7_Templates := "SrcType := Int" } EQ_Contact(in1 := "IEC_Counter_0_DB[1]".CV, in2 := 0)
      Move(in := 128, out1 => "Emitter_Part")
   END_RUNG
   RUNG wire#powerrail
      { S7_Templates := "SrcType := Int" } EQ_Contact(in1 := "IEC_Counter_0_DB[1]".CV, in2 := 1)
      Move(in := 256, out1 => "Emitter_Part")
   END_RUNG
   RUNG wire#powerrail
      { S7_Templates := "SrcType := Int" } EQ_Contact(in1 := "IEC_Counter_0_DB[1]".CV, in2 := 2)
      Move(in := 512, out1 => "Emitter_Part")
   END_RUNG
   RUNG wire#powerrail
      { S7_Templates := "SrcType := Int" } EQ_Contact(in1 := "IEC_Counter_0_DB[1]".CV, in2 := 3)
      Move(in := 1024, out1 => "Emitter_Part")
   END_RUNG
   RUNG wire#powerrail
      { S7_Templates := "SrcType := Int" } EQ_Contact(in1 := "IEC_Counter_0_DB[1]".CV, in2 := 4)
      Move(in := 2048, out1 => "Emitter_Part")
   END_RUNG
   RUNG wire#powerrail
      { S7_Templates := "SrcType := Int" } EQ_Contact(in1 := "IEC_Counter_0_DB[1]".CV, in2 := 5)
      Move(in := 4096, out1 => "Emitter_Part")
   END_RUNG
   // the same network as SCL:
   IF "IEC_Counter_0_DB[1]".CV = 0 THEN "Emitter_Part" := 128; END_IF;
   IF "IEC_Counter_0_DB[1]".CV = 1 THEN "Emitter_Part" := 256; END_IF;
   IF "IEC_Counter_0_DB[1]".CV = 2 THEN "Emitter_Part" := 512; END_IF;
   IF "IEC_Counter_0_DB[1]".CV = 3 THEN "Emitter_Part" := 1024; END_IF;
   IF "IEC_Counter_0_DB[1]".CV = 4 THEN "Emitter_Part" := 2048; END_IF;
   IF "IEC_Counter_0_DB[1]".CV = 5 THEN "Emitter_Part" := 4096; END_IF;
END_REGION

REGION Network 16: Emitter Trigger
   RUNG wire#powerrail
      I_Contact( "Stop Sensor 1" )
      wire#w1
      Coil( "Emitter_Emit" )
   END_RUNG
   RUNG wire#powerrail
      I_Contact( "Stop Sensor 2" )
   END_RUNG wire#w1
   // the same network as SCL:
   "Emitter_Emit" := NOT "Stop Sensor 1" OR NOT "Stop Sensor 2";
END_REGION

REGION Network 17
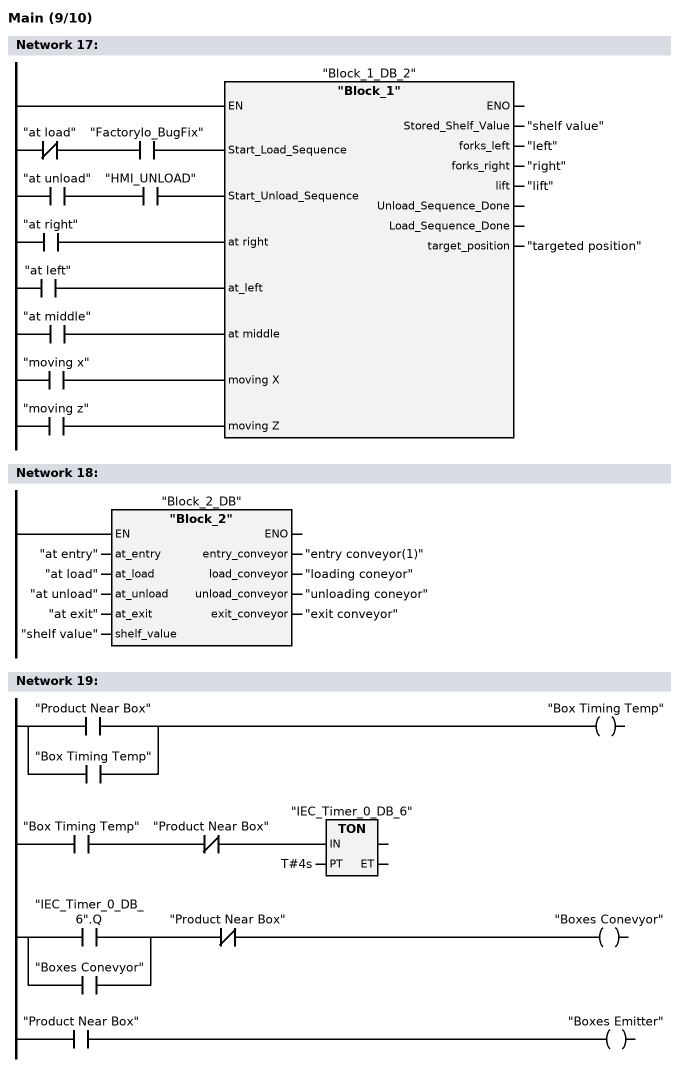
   RUNG wire#powerrail
      "Block_1_DB_2"(Start_Load_Sequence := wire#w1, Start_Unload_Sequence := wire#w2, "at right" := wire#w3, at_left := wire#w4, "at middle" := wire#w5, "moving X" := wire#w6, "moving Z" := wire#w7, Stored_Shelf_Value => "shelf value", forks_left => "left", forks_right => "right", lift => "lift", Unload_Sequence_Done =>, Load_Sequence_Done =>, target_position => "targeted position")
   END_RUNG
   RUNG wire#powerrail
      I_Contact( "at load" )
      Contact( "FactoryIo_BugFix" )
   END_RUNG wire#w1
   RUNG wire#powerrail
      Contact( "at unload" )
      Contact( "HMI_UNLOAD" )
   END_RUNG wire#w2
   RUNG wire#powerrail
      Contact( "at right" )
   END_RUNG wire#w3
   RUNG wire#powerrail
      Contact( "at left" )
   END_RUNG wire#w4
   RUNG wire#powerrail
      Contact( "at middle" )
   END_RUNG wire#w5
   RUNG wire#powerrail
      Contact( "moving x" )
   END_RUNG wire#w6
   RUNG wire#powerrail
      Contact( "moving z" )
   END_RUNG wire#w7
   // the same network as SCL:
   "Block_1_DB_2"(Start_Load_Sequence := NOT "at load" AND "FactoryIo_BugFix",   // "Block_1"
                  Start_Unload_Sequence := "at unload" AND "HMI_UNLOAD",
                  "at right" := "at right",
                  at_left := "at left",
                  "at middle" := "at middle",
                  "moving X" := "moving x",
                  "moving Z" := "moving z",
                  Stored_Shelf_Value => "shelf value",
                  forks_left => "left",
                  forks_right => "right",
                  lift => "lift",
                  target_position => "targeted position");
END_REGION

REGION Network 18
   RUNG wire#powerrail
      "Block_2_DB"(at_entry := "at entry", at_load := "at load", at_unload := "at unload", at_exit := "at exit", shelf_value := "shelf value", entry_conveyor => "entry conveyor(1)", load_conveyor => "loading coneyor", unload_conveyor => "unloading coneyor", exit_conveyor => "exit conveyor")
   END_RUNG
   // the same network as SCL:
   "Block_2_DB"(at_entry := "at entry",   // "Block_2"
                at_load := "at load",
                at_unload := "at unload",
                at_exit := "at exit",
                shelf_value := "shelf value",
                entry_conveyor => "entry conveyor(1)",
                load_conveyor => "loading coneyor",
                unload_conveyor => "unloading coneyor",
                exit_conveyor => "exit conveyor");
END_REGION

REGION Network 19
   "Box Timing Temp" := "Product Near Box" OR "Box Timing Temp";
   "IEC_Timer_0_DB_6".TON(IN := "Box Timing Temp" AND NOT "Product Near Box", PT := T#4s);
   "Boxes Conevyor" := ("IEC_Timer_0_DB_6".Q OR "Boxes Conevyor") AND NOT "Product Near Box";
   "Boxes Emitter" := "Product Near Box";
END_REGION

REGION Network 20
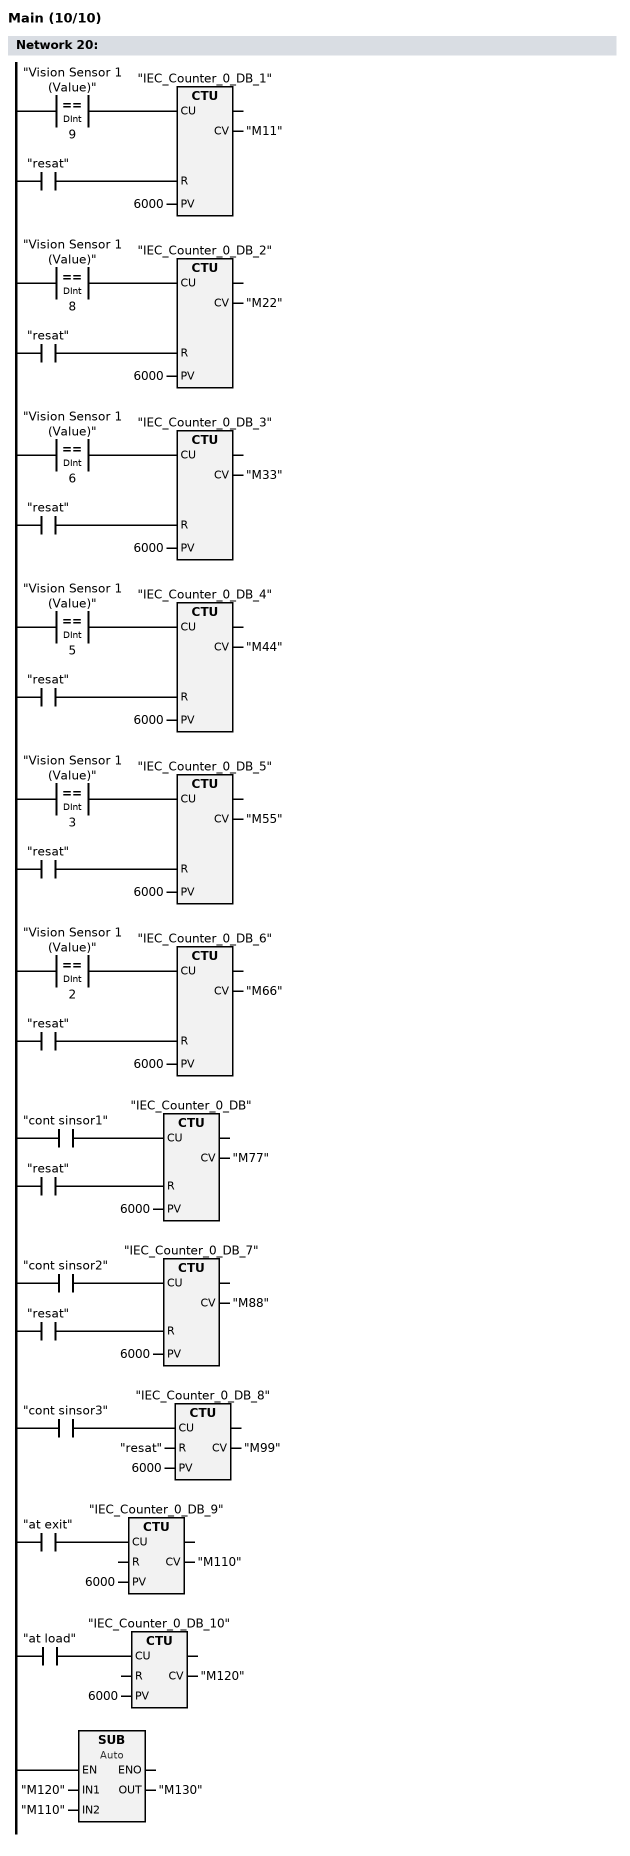
   "IEC_Counter_0_DB_1".CTU(CU := "Vision Sensor 1 (Value)" = 9, R := "resat", PV := 6000, CV => "M11");
   "IEC_Counter_0_DB_2".CTU(CU := "Vision Sensor 1 (Value)" = 8, R := "resat", PV := 6000, CV => "M22");
   "IEC_Counter_0_DB_3".CTU(CU := "Vision Sensor 1 (Value)" = 6, R := "resat", PV := 6000, CV => "M33");
   "IEC_Counter_0_DB_4".CTU(CU := "Vision Sensor 1 (Value)" = 5, R := "resat", PV := 6000, CV => "M44");
   "IEC_Counter_0_DB_5".CTU(CU := "Vision Sensor 1 (Value)" = 3, R := "resat", PV := 6000, CV => "M55");
   "IEC_Counter_0_DB_6".CTU(CU := "Vision Sensor 1 (Value)" = 2, R := "resat", PV := 6000, CV => "M66");
   "IEC_Counter_0_DB".CTU(CU := "cont sinsor1", R := "resat", PV := 6000, CV => "M77");
   "IEC_Counter_0_DB_7".CTU(CU := "cont sinsor2", R := "resat", PV := 6000, CV => "M88");
   "IEC_Counter_0_DB_8".CTU(CU := "cont sinsor3", R := "resat", PV := 6000, CV => "M99");
   "IEC_Counter_0_DB_9".CTU(CU := "at exit", PV := 6000, CV => "M110");
   "IEC_Counter_0_DB_10".CTU(CU := "at load", PV := 6000, CV => "M120");
   "M130" := "M120" - "M110";
END_REGION
END_ORGANIZATION_BLOCK

(* ===== HMI "HMI_RT_1" =====
system functions are stored by id; their names below are inferred from use
connection "HMI_Connection_1": ETHERNET, S7_1200_OMS

HMI tags "Default tag table"
   "Tag_ScreenNumber" : UInt, internal
   "M11" : DInt = PLC M11 AT %MD60, 1 s
   "M22" : DInt = PLC M22 AT %MD64, 1 s
   "M33" : DInt = PLC M33 AT %MD68, 1 s
   "M44" : DInt = PLC M44 AT %MD72, 1 s
   "M55" : DInt = PLC M55 AT %MD76, 1 s
   "M66" : DInt = PLC M66 AT %MD80, 1 s
   "shelf value" : Word = PLC "shelf value" AT %MW46, 1 s
   "M77" : DInt = PLC M77 AT %MD88, 1 s
   "M88" : DInt = PLC M88 AT %MD92, 1 s
   "M99" : DInt = PLC M99 AT %MD96, 1 s
   "resat" : Bool = PLC resat AT %M100.0, 1 s
   "at unload" : Bool = PLC "at unload" AT %I13.7, 1 s
   "M110" : DInt = PLC M110 AT %MD110, 1 s
   "M120" : DInt = PLC M120 AT %MD114, 1 s
   "M130" : DInt = PLC M130 AT %MD118, 1 s
   "HMI_UNLOAD" : Bool = PLC HMI_UNLOAD AT %I122.0, 1 s

screen "Root screen" 1280x740, template "Template_1"
   on GenerateScreen: SetTag("Tag_ScreenNumber", 1)
   TextField "HmiScreenItemData_2" at 128,324 size 1024x27; Text 'Welcome to HMI_1 (TP1200 Comfort)!'
   Button "HmiScreenItemData" at 36,36 size 159x47; TextOff 'control'; TextOn 'Screen0'; PictureOff "Navigates to Screen0 for TP1200 Comfort 15.1.0.0"; PictureOn "Navigates to Screen0 for TP1200 Comfort 15.1.0.0"
      on Release: ActivateScreen("Screen0", 0)
   Button "HmiScreenItemData_3" at 36,87 size 159x47; TextOff 'System screens'; PictureOff "Navigates to System screens for TP1200 Comfort 15.1.0.0"; PictureOn "Navigates to System screens for TP1200 Comfort 15.1.0.0"
      on Release: ActivateScreen("System screens", 0)

Template "Template_1" 1280x740
   Button "Exit" at 1200,679 size 78x59; TextOff 'Exit'; PictureOff "ExitRuntime_TP1200_Comfort_TR"; PictureOn "ExitRuntime_TP1200_Comfort_TR"
      on Release: StopRuntime(0)
   Button "Log on" at 1120,679 size 78x59; TextOff 'Log on'; PictureOff "Login_TP1200_Comfort_TR"; PictureOn "Login_TP1200_Comfort_TR"
      on Release: function_a2a04561()
   Button "Language" at 1040,679 size 78x59; TextOff 'Language'; PictureOff "ToggleLanguage_TP1200_Comfort_TR"; PictureOn "ToggleLanguage_TP1200_Comfort_TR"
      on Release: function_fb9197e8(-1)
   Button "Template_Button" at 960,679 size 78x59; TextOff 'Text'
   Button "Template_Button_1" at 880,679 size 78x59; TextOff 'Text'
   Button "Template_Button_2" at 800,679 size 78x59; TextOff 'Text'
   Button "Template_Button_3" at 720,679 size 78x59; TextOff 'Text'
   Button "Template_Button_4" at 640,679 size 78x59; TextOff 'Text'
   Button "Template_Button_5" at 561,679 size 78x59; TextOff 'Text'
   Button "Template_Button_6" at 481,679 size 78x59; TextOff 'Text'
   Button "Template_Button_7" at 401,679 size 78x59; TextOff 'Text'
   Button "Template_Button_8" at 321,679 size 78x59; TextOff 'Text'
   Button "Template_Button_9" at 241,679 size 78x59; TextOff 'Text'
   Button "Template_Button_10" at 161,679 size 78x59; TextOff 'Text'
   Button "Template_Button_11" at 81,679 size 78x59; TextOff 'Text'
   Button "Start screen" at 1,679 size 78x59; TextOff 'Start screen'; PictureOff "NavigateHome_TP1200_Comfort_TR"; PictureOn "NavigateHome_TP1200_Comfort_TR"
      on Release: ActivateScreen("Root screen", 0)

screen "Screen0" 1280x740, template "Template_1"
   on GenerateScreen: SetTag("Tag_ScreenNumber", 2)
   TextField "HmiScreenItemData" at 84,11 size 1024x27; Text 'cntrol'
   Button "Back" at 1,1 size 159x47; TextOff 'Back'
      on Release: ActivateScreen("Root screen", 0)
   IOField "I/O field_1" at 157,155 size 195x72; FormatPattern s9999999999
      ProcessValue <- "M11"
   IOField "I/O field_2" at 161,77 size 195x69; FormatPattern s9999999999
      ProcessValue <- "M22"
   IOField "I/O field_3" at 553,111 size 203x92; FormatPattern 9999999
      ProcessValue <- "M77"
   IOField "I/O field_4" at 160,289 size 196x72; FormatPattern s9999999999
      ProcessValue <- "M33"
   IOField "I/O field_5" at 157,369 size 196x70; FormatPattern s9999999999
      ProcessValue <- "M44"
   IOField "I/O field_6" at 546,320 size 207x93; FormatPattern s9999999999
      ProcessValue <- "M88"
   IOField "I/O field_7" at 157,565 size 196x61; FormatPattern s9999999999
      ProcessValue <- "M55"
   IOField "I/O field_8" at 157,495 size 196x66; FormatPattern s9999999999
      ProcessValue <- "M66"
   IOField "I/O field_9" at 549,511 size 207x85; FormatPattern s9999999999
      ProcessValue <- "M99"
   IOField "I/O field_10" at 973,285 size 301x158; FormatPattern s9999999999
      ProcessValue <- "M130"
   Button "Button_1" at 18,76 size 129x61; TextOff 'Black part A'
   Button "Button_2" at 15,165 size 133x61; TextOff 'Black part B'
   Button "Button_3" at 791,318 size 171x90; TextOff 'the warehouse'
   Button "Button_4" at 371,129 size 167x55; TextOff 'Assembled Black'
   Button "Button_5" at 369,331 size 163x59; TextOff 'Assembled Green'
   Button "Button_6" at 368,520 size 165x57; TextOff 'Assembled Blue'
   Button "Button_7" at 15,295 size 133x60; TextOff 'Green part A'
   Button "Button_8" at 18,382 size 127x60; TextOff 'Green part B'
   Button "Button_9" at 15,495 size 124x60; TextOff 'Blue part A'
   Button "Button_10" at 18,573 size 124x50; TextOff 'Blue part B'
   Switch "Pushbutton_Square_N_Mono" at 1026,36 size 200x50; CaptionText 'Switch'; TextOff 'resat / 0'; TextOn 'resat / 1'; PictureOff "Pushbutton_Square_N_Off_mono"; PictureOn "Pushbutton_Square_N_On_mono"
      ProcessValue <- "resat"
   Switch "Pushbutton_Square_N_Mono_1" at 1017,100 size 213x108; CaptionText 'Switch'; TextOff 'Unload / 0'; TextOn 'Unload / 1'; PictureOff "Pushbutton_Square_N_Off_mono"; PictureOn "Pushbutton_Square_N_On_mono"
      ProcessValue <- "HMI_UNLOAD"

screen "Screen1" 1280x740, template "Template_1"
   on GenerateScreen: SetTag("Tag_ScreenNumber", 3)
   TextField "HmiScreenItemData" at 128,324 size 1024x27; Text 'Screen1'
   Button "Back" at 1,1 size 159x47; TextOff 'Back'
      on Release: ActivateScreen("Root screen", 0)

screen "System screens" 1280x740, template "Template_1"
   on GenerateScreen: SetTag("Tag_ScreenNumber", 4)
   Button "Back" at 1,1 size 159x47; TextOff 'Back'
      on Release: ActivateScreen("Root screen", 0)
   Button "HmiScreenItemData" at 36,95 size 159x47; TextOff 'SIMATIC PLC system diagnos...'; PictureOff "Navigates to SIMATIC PLC system diagnostics for TP1200 Comfort 15.1.0.0"; PictureOn "Navigates to SIMATIC PLC system diagnostics for TP1200 Comfort 15.1.0.0"
      on Release: ActivateScreen("SIMATIC PLC system diagnostics", 0)
   Button "HmiScreenItemData_1" at 36,154 size 159x47; TextOff 'Project information'; PictureOff "Navigates to Project information for TP1200 Comfort 15.1.0.0"; PictureOn "Navigates to Project information for TP1200 Comfort 15.1.0.0"
      on Release: ActivateScreen("Project information", 0)
   Button "HmiScreenItemData_2" at 36,213 size 159x47; TextOff 'System settings'; PictureOff "Navigates to System settings for TP1200 Comfort 15.1.0.0"; PictureOn "Navigates to System settings for TP1200 Comfort 15.1.0.0"
      on Release: ActivateScreen("System settings", 0)
   Button "HmiScreenItemData_3" at 36,272 size 159x47; TextOff 'User administration'; PictureOff "Navigates to User administration for TP1200 Comfort 15.1.0.0"; PictureOn "Navigates to User administration for TP1200 Comfort 15.1.0.0"
      on Release: ActivateScreen("User administration", 0)
   Button "HmiScreenItemData_4" at 36,331 size 159x47; TextOff 'System information'; PictureOff "Navigates to System information for TP1200 Comfort 15.1.0.0"; PictureOn "Navigates to System information for TP1200 Comfort 15.1.0.0"
      on Release: ActivateScreen("System information", 0)
   Button "HmiScreenItemData_5" at 36,390 size 159x47; TextOff 'Different jobs'; PictureOff "Navigates to Different jobs for TP1200 Comfort 15.1.0.0"; PictureOn "Navigates to Different jobs for TP1200 Comfort 15.1.0.0"
      on Release: ActivateScreen("Different jobs", 0)

screen "SIMATIC PLC system diagnostics" 1280x740, template "Template_1"
   on GenerateScreen: SetTag("Tag_ScreenNumber", 5)
   SysDiagControl "HmiScreenItemData" at 1,49 size 1276x623
   Button "Back" at 1,1 size 159x47; TextOff 'Back'
      on Release: ActivateScreen("System screens", 0)

screen "Project information" 1280x740, template "Template_1"
   on GenerateScreen: SetTag("Tag_ScreenNumber", 6)
   TextField "HmiScreenItemData" at 35,51 size 171x28; Text 'Project name:'
   TextField "HmiScreenItemData_1" at 241,51 size 1004x28; Text 'FactoryIO_Template_S7-1200_V15_V15.1'
   TextField "HmiScreenItemData_2" at 35,81 size 171x28; Text 'Created on:'
   TextField "HmiScreenItemData_3" at 241,81 size 1004x28; Text '4/7/2016 12:51:36 PM'
   TextField "HmiScreenItemData_4" at 35,111 size 171x28; Text 'Author:'
   TextField "HmiScreenItemData_5" at 241,111 size 1004x28; Text 'ayman'
   TextField "HmiScreenItemData_6" at 35,141 size 171x28; Text 'Description:'
   TextField "HmiScreenItemData_7" at 241,141 size 1004x28; Text '(not configured)'
   Button "Back" at 1,1 size 159x47; TextOff 'Back'
      on Release: ActivateScreen("System screens", 0)

screen "System settings" 1280x740, template "Template_1"
   on GenerateScreen: SetTag("Tag_ScreenNumber", 7)
   Button "Calibrate screen" at 36,95 size 159x47; TextOff 'Calibrate screen'
      on Release: function_bc3e350c()
   Button "Clean screen" at 36,154 size 159x47; TextOff 'Clean screen'
      on Release: function_be740847(30)
   Button "Back" at 1,1 size 159x47; TextOff 'Back'
      on Release: ActivateScreen("System screens", 0)

screen "User administration" 1280x740, template "Template_1"
   on GenerateScreen: SetTag("Tag_ScreenNumber", 8)
   UserView "HmiScreenItemData" at 1,49 size 1276x623
   Button "Back" at 1,1 size 159x47; TextOff 'Back'
      on Release: ActivateScreen("System screens", 0)

screen "System information" 1280x740, template "Template_1"
   on GenerateScreen: SetTag("Tag_ScreenNumber", 9)
   TextField "HmiScreenItemData" at 35,51 size 171x28; Text 'HMI device type:'
   TextField "HmiScreenItemData_1" at 241,51 size 1004x28; Text 'TP1200 Comfort 15.1.0.0'
   TextField "HmiScreenItemData_2" at 35,81 size 171x28; Text 'Version:'
   TextField "HmiScreenItemData_3" at 35,111 size 171x28; Text 'Connection:'
   TextField "HmiScreenItemData_4" at 241,111 size 1004x28; Text 'ETHERNET'
   TextField "HmiScreenItemData_5" at 35,141 size 171x28; Text 'PLC:'
   TextField "HmiScreenItemData_6" at 241,141 size 1004x28; Text 'SIMATIC S7 1200'
   Button "Display version" at 241,81 size 1004x28; TextOff 'Display version'
      on Release: function_febcb963(-1)
   Button "Back" at 1,1 size 159x47; TextOff 'Back'
      on Release: ActivateScreen("System screens", 0)

screen "Different jobs" 1280x740, template "Template_1"
   on GenerateScreen: SetTag("Tag_ScreenNumber", 10)
   Button "Online" at 36,95 size 159x47; TextOff 'Online'
      on Release: function_bb44b551(0)
   Button "Offline" at 36,154 size 159x47; TextOff 'Offline'
      on Release: function_bb44b551(1)
   Button "Transfer" at 36,213 size 159x47; TextOff 'Transfer'
      on Release: function_bb44b551(2)
   Button "Toggle language" at 36,272 size 159x47; TextOff 'Toggle language'
      on Release: function_fb9197e8(-1)
   Button "Control Panel" at 36,331 size 159x47; TextOff 'Control Panel'
      on Release: function_f34a74f3()
   Button "Stop Runtime" at 36,390 size 159x47; TextOff 'Stop Runtime'
      on Release: StopRuntime(0)
   Button "Back" at 1,1 size 159x47; TextOff 'Back'
      on Release: ActivateScreen("System screens", 0)
*)